LIN {X 0,Y 323.294,Z 676.092,A -85,B 0,C 180,E1 15567.964,E2 15567.964} C_VEL
LIN {X 0,Y 321.355,Z 689.746,A -85,B 0,C 180,E1 15566.345,E2 15566.345} C_VEL
LIN {X 0,Y 319.343,Z 702.477,A -85,B 0,C 180,E1 15564.432,E2 15564.432} C_VEL
LIN {X 0,Y 317.522,Z 713.237,A -85,B 0,C 180,E1 15562.402,E2 15562.402} C_VEL
LIN {X 0,Y 315.747,Z 723.463,A -85,B 0,C 180,E1 15559.972,E2 15559.972} C_VEL
LIN {X 0,Y 314.38,Z 731.614,A -85,B 0,C 180,E1 15557.512,E2 15557.512} C_VEL
LIN {X 0,Y 313.266,Z 738.806,A -85,B 0,C 180,E1 15554.64,E2 15554.64} C_VEL
LIN {X 0,Y 312.607,Z 743.939,A -85,B 0,C 180,E1 15551.797,E2 15551.797} C_VEL
LIN {X 0,Y 312.265,Z 747.451,A -85,B 0,C 180,E1 15548.715,E2 15548.715} C_VEL
LIN {X 0,Y 312.168,Z 749.028,A -85,B 0,C 180,E1 15545.799,E2 15545.799} C_VEL
LIN {X 0,Y 312.206,Z 748.828,A -85,B 0,C 180,E1 15542.747,E2 15542.747} C_VEL
LIN {X 0,Y 312.438,Z 746.912,A -85,B 0,C 180,E1 15539.776,E2 15539.776} C_VEL
LIN {X 0,Y 312.956,Z 743.159,A -85,B 0,C 180,E1 15536.833,E2 15536.833} C_VEL
LIN {X 0,Y 313.904,Z 737.534,A -85,B 0,C 180,E1 15533.898,E2 15533.898} C_VEL
LIN {X 0,Y 315.295,Z 730.063,A -85,B 0,C 180,E1 15531.108,E2 15531.108} C_VEL
LIN {X 0,Y 316.967,Z 721.566,A -85,B 0,C 180,E1 15528.658,E2 15528.658} C_VEL
LIN {X 0,Y 319.018,Z 711.003,A -85,B 0,C 180,E1 15526.287,E2 15526.287} C_VEL
LIN {X 0,Y 321.176,Z 699.388,A -85,B 0,C 180,E1 15524.215,E2 15524.215} C_VEL
LIN {X 0,Y 323.403,Z 686.141,A -85,B 0,C 180,E1 15522.365,E2 15522.365} C_VEL
LIN {X 0,Y 325.505,Z 671.84,A -85,B 0,C 180,E1 15520.801,E2 15520.801} C_VEL
LIN {X 0,Y 327.265,Z 657.03,A -85,B 0,C 180,E1 15519.581,E2 15519.581} C_VEL
LIN {X 0,Y 328.688,Z 641.061,A -85,B 0,C 180,E1 15518.618,E2 15518.618} C_VEL
LIN {X 0,Y 329.594,Z 624.254,A -85,B 0,C 180,E1 15517.968,E2 15517.968} C_VEL
LIN {X 0,Y 333.422,Z 501.812,A -85,B 0,C 180,E1 15515.207,E2 15515.207} C_VEL
LIN {X 0,Y 331.425,Z 482.705,A -85,B 0,C 180,E1 15514.449,E2 15514.449} C_VEL
LIN {X 0,Y 335.442,Z 437.528,A -85,B 0,C 180,E1 15509.848,E2 15509.848} C_VEL
LIN {X 0,Y 338.999,Z 399.053,A -85,B 0,C 180,E1 15505.967,E2 15505.967} C_VEL
LIN {X 0,Y 342.306,Z 362.127,A -85,B 0,C 180,E1 15502.249,E2 15502.249} C_VEL
LIN {X 0,Y 337.591,Z 346.974,A -85,B 0,C 180,E1 15499.734,E2 15499.734} C_VEL
LIN {X 0,Y 332.324,Z 333.278,A -85,B 0,C 180,E1 15497.149,E2 15497.149} C_VEL
LIN {X 0,Y 326.437,Z 320.297,A -85,B 0,C 180,E1 15494.366,E2 15494.366} C_VEL
LIN {X 0,Y 321.45,Z 310.966,A -85,B 0,C 180,E1 15492.029,E2 15492.029} C_VEL
LIN {X 0,Y 319.417,Z 307.063,A -85,B 0,C 180,E1 15491.009,E2 15491.009} C_VEL
LIN {X 0,Y 317.338,Z 303.417,A -85,B 0,C 180,E1 15489.98,E2 15489.98} C_VEL
LIN {X 0,Y 316.226,Z 301.786,A -85,B 0,C 180,E1 15489.464,E2 15489.464} C_VEL
LIN {X 0,Y 314.376,Z 298.507,A -85,B 0,C 180,E1 15488.478,E2 15488.478} C_VEL
LIN {X 0,Y 314.155,Z 297.393,A -85,B 0,C 180,E1 15487.959,E2 15487.959} C_VEL
LIN {X 0,Y 314.165,Z 297.347,A -85,B 0,C 180,E1 15483.467,E2 15483.467} C_VEL
LIN {X 0,Y 314.171,Z 297.344,A -85,B 0,C 180,E1 15479.089,E2 15479.089} C_VEL
LIN {X 0,Y 314.151,Z 297.354,A -85,B 0,C 180,E1 15474.522,E2 15474.522} C_VEL
LIN {X 0,Y 314.146,Z 297.345,A -85,B 0,C 180,E1 15470.104,E2 15470.104} C_VEL
LIN {X 0,Y 314.161,Z 297.354,A -85,B 0,C 180,E1 15465.627,E2 15465.627} C_VEL
LIN {X 0,Y 314.17,Z 297.343,A -85,B 0,C 180,E1 15461.251,E2 15461.251} C_VEL
LIN {X 0,Y 314.172,Z 297.351,A -85,B 0,C 180,E1 15456.758,E2 15456.758} C_VEL
LIN {X 0,Y 314.155,Z 297.349,A -85,B 0,C 180,E1 15452.22,E2 15452.22} C_VEL
LIN {X 0,Y 314.207,Z 297.632,A -85,B 0,C 180,E1 15448.543,E2 15448.543} C_VEL
LIN {X 0,Y 315.623,Z 301.081,A -85,B 0,C 180,E1 15447.631,E2 15447.631} C_VEL
LIN {X 0,Y 322.969,Z 317.218,A -85,B 0,C 180,E1 15443.751,E2 15443.751} C_VEL
LIN {X 0,Y 325.12,Z 321.958,A -85,B 0,C 180,E1 15442.766,E2 15442.766} C_VEL
LIN {X 0,Y 339.923,Z 346.539,A -85,B 0,C 180,E1 15439.593,E2 15439.593} C_VEL
LIN {X 0,Y 354.859,Z 373.04,A -85,B 0,C 180,E1 15436.679,E2 15436.679} C_VEL
LIN {X 0,Y 356.871,Z 377.15,A -85,B 0,C 180,E1 15436.291,E2 15436.291} C_VEL
LIN {X 0,Y 344.034,Z 576.734,A -85,B 0,C 180,E1 15431.093,E2 15431.093} C_VEL
LIN {X 0,Y 341.881,Z 598.232,A -85,B 0,C 180,E1 15430.243,E2 15430.243} C_VEL
LIN {X 0,Y 339.198,Z 619.151,A -85,B 0,C 180,E1 15429.107,E2 15429.107} C_VEL
LIN {X 0,Y 336.079,Z 639.65,A -85,B 0,C 180,E1 15427.655,E2 15427.655} C_VEL
LIN {X 0,Y 332.807,Z 658.657,A -85,B 0,C 180,E1 15425.966,E2 15425.966} C_VEL
LIN {X 0,Y 329.239,Z 677.46,A -85,B 0,C 180,E1 15423.908,E2 15423.908} C_VEL
LIN {X 0,Y 325.708,Z 695.046,A -85,B 0,C 180,E1 15421.558,E2 15421.558} C_VEL
LIN {X 0,Y 322.353,Z 711.252,A -85,B 0,C 180,E1 15418.936,E2 15418.936} C_VEL
LIN {X 0,Y 319.275,Z 726.233,A -85,B 0,C 180,E1 15416.001,E2 15416.001} C_VEL
LIN {X 0,Y 316.82,Z 738.788,A -85,B 0,C 180,E1 15413.035,E2 15413.035} C_VEL
LIN {X 0,Y 314.859,Z 749.859,A -85,B 0,C 180,E1 15409.861,E2 15409.861} C_VEL
LIN {X 0,Y 313.501,Z 758.929,A -85,B 0,C 180,E1 15406.679,E2 15406.679} C_VEL
LIN {X 0,Y 312.614,Z 766.626,A -85,B 0,C 180,E1 15403.312,E2 15403.312} C_VEL
LIN {X 0,Y 312.189,Z 772.809,A -85,B 0,C 180,E1 15399.771,E2 15399.771} C_VEL
LIN {X 0,Y 312.1,Z 776.968,A -85,B 0,C 180,E1 15396.436,E2 15396.436} C_VEL
LIN {X 0,Y 312.119,Z 779.473,A -85,B 0,C 180,E1 15393.12,E2 15393.12} C_VEL
LIN {X 0,Y 312.146,Z 780.41,A -85,B 0,C 180,E1 15389.814,E2 15389.814} C_VEL
LIN {X 0,Y 312.083,Z 779.858,A -85,B 0,C 180,E1 15386.508,E2 15386.508} C_VEL
LIN {X 0,Y 312.051,Z 777.77,A -85,B 0,C 180,E1 15383.189,E2 15383.189} C_VEL
LIN {X 0,Y 312.18,Z 774.12,A -85,B 0,C 180,E1 15379.852,E2 15379.852} C_VEL
LIN {X 0,Y 312.695,Z 768.613,A -85,B 0,C 180,E1 15376.311,E2 15376.311} C_VEL
LIN {X 0,Y 313.732,Z 761.756,A -85,B 0,C 180,E1 15372.948,E2 15372.948} C_VEL
LIN {X 0,Y 315.522,Z 752.593,A -85,B 0,C 180,E1 15369.404,E2 15369.404} C_VEL
LIN {X 0,Y 318.153,Z 741.278,A -85,B 0,C 180,E1 15365.884,E2 15365.884} C_VEL
LIN {X 0,Y 321.514,Z 728.328,A -85,B 0,C 180,E1 15362.595,E2 15362.595} C_VEL
LIN {X 0,Y 325.509,Z 713.816,A -85,B 0,C 180,E1 15359.546,E2 15359.546} C_VEL
LIN {X 0,Y 330.18,Z 697.464,A -85,B 0,C 180,E1 15356.697,E2 15356.697} C_VEL
LIN {X 0,Y 335.464,Z 679.029,A -85,B 0,C 180,E1 15354.042,E2 15354.042} C_VEL
LIN {X 0,Y 340.919,Z 659.877,A -85,B 0,C 180,E1 15351.768,E2 15351.768} C_VEL
LIN {X 0,Y 346.959,Z 638.42,A -85,B 0,C 180,E1 15349.686,E2 15349.686} C_VEL
LIN {X 0,Y 353.072,Z 616.191,A -85,B 0,C 180,E1 15347.951,E2 15347.951} C_VEL
LIN {X 0,Y 358.873,Z 594.337,A -85,B 0,C 180,E1 15346.623,E2 15346.623} C_VEL
LIN {X 0,Y 364.618,Z 570.64,A -85,B 0,C 180,E1 15345.534,E2 15345.534} C_VEL
LIN {X 0,Y 377.031,Z 516.92,A -85,B 0,C 180,E1 15343.532,E2 15343.532} C_VEL
LIN {X 0,Y 381.467,Z 500.047,A -85,B 0,C 180,E1 15342.895,E2 15342.895} C_VEL
LIN {X 0,Y 366.445,Z 559.755,A -85,B 0,C 180,E1 15340.585,E2 15340.585} C_VEL
LIN {X 0,Y 360.935,Z 581.963,A -85,B 0,C 180,E1 15339.579,E2 15339.579} C_VEL
LIN {X 0,Y 355.075,Z 603.113,A -85,B 0,C 180,E1 15338.279,E2 15338.279} C_VEL
LIN {X 0,Y 348.859,Z 624.354,A -85,B 0,C 180,E1 15336.594,E2 15336.594} C_VEL
LIN {X 0,Y 342.955,Z 643.935,A -85,B 0,C 180,E1 15334.646,E2 15334.646} C_VEL
LIN {X 0,Y 337.175,Z 662.515,A -85,B 0,C 180,E1 15332.361,E2 15332.361} C_VEL
LIN {X 0,Y 331.809,Z 679.598,A -85,B 0,C 180,E1 15329.788,E2 15329.788} C_VEL
LIN {X 0,Y 327.161,Z 694.304,A -85,B 0,C 180,E1 15327.088,E2 15327.088} C_VEL
LIN {X 0,Y 323.006,Z 707.545,A -85,B 0,C 180,E1 15324.117,E2 15324.117} C_VEL
LIN {X 0,Y 319.633,Z 718.492,A -85,B 0,C 180,E1 15321.083,E2 15321.083} C_VEL
LIN {X 0,Y 316.864,Z 727.897,A -85,B 0,C 180,E1 15317.823,E2 15317.823} C_VEL
LIN {X 0,Y 314.86,Z 735.32,A -85,B 0,C 180,E1 15314.528,E2 15314.528} C_VEL
LIN {X 0,Y 313.523,Z 740.919,A -85,B 0,C 180,E1 15311.217,E2 15311.217} C_VEL
LIN {X 0,Y 312.721,Z 744.807,A -85,B 0,C 180,E1 15307.902,E2 15307.902} C_VEL
LIN {X 0,Y 312.307,Z 747.109,A -85,B 0,C 180,E1 15304.406,E2 15304.406} C_VEL
LIN {X 0,Y 312.167,Z 747.631,A -85,B 0,C 180,E1 15301.101,E2 15301.101} C_VEL
LIN {X 0,Y 312.123,Z 746.506,A -85,B 0,C 180,E1 15297.796,E2 15297.796} C_VEL
LIN {X 0,Y 312.205,Z 743.731,A -85,B 0,C 180,E1 15294.486,E2 15294.486} C_VEL
LIN {X 0,Y 312.502,Z 739.236,A -85,B 0,C 180,E1 15291.165,E2 15291.165} C_VEL
LIN {X 0,Y 313.109,Z 733.292,A -85,B 0,C 180,E1 15288.02,E2 15288.02} C_VEL
LIN {X 0,Y 314.157,Z 725.57,A -85,B 0,C 180,E1 15284.871,E2 15284.871} C_VEL
LIN {X 0,Y 315.737,Z 715.857,A -85,B 0,C 180,E1 15281.728,E2 15281.728} C_VEL
LIN {X 0,Y 317.776,Z 704.613,A -85,B 0,C 180,E1 15278.786,E2 15278.786} C_VEL
LIN {X 0,Y 320.217,Z 691.886,A -85,B 0,C 180,E1 15276.051,E2 15276.051} C_VEL
LIN {X 0,Y 322.985,Z 677.669,A -85,B 0,C 180,E1 15273.526,E2 15273.526} C_VEL
LIN {X 0,Y 325.992,Z 661.889,A -85,B 0,C 180,E1 15271.213,E2 15271.213} C_VEL
LIN {X 0,Y 329.153,Z 644.286,A -85,B 0,C 180,E1 15269.111,E2 15269.111} C_VEL
LIN {X 0,Y 332.082,Z 626.513,A -85,B 0,C 180,E1 15267.387,E2 15267.387} C_VEL
LIN {X 0,Y 334.806,Z 607.979,A -85,B 0,C 180,E1 15265.947,E2 15265.947} C_VEL
LIN {X 0,Y 337.196,Z 588.684,A -85,B 0,C 180,E1 15264.778,E2 15264.778} C_VEL
LIN {X 0,Y 339.329,Z 567.504,A -85,B 0,C 180,E1 15263.841,E2 15263.841} C_VEL
LIN {X 0,Y 341.441,Z 536.028,A -85,B 0,C 180,E1 15262.91,E2 15262.91} C_VEL
LIN {X 0,Y 351.309,Z 385.374,A -85,B 0,C 180,E1 15258.813,E2 15258.813} C_VEL
LIN {X 0,Y 349.678,Z 373.169,A -85,B 0,C 180,E1 15258.18,E2 15258.18} C_VEL
LIN {X 0,Y 335.154,Z 345.914,A -85,B 0,C 180,E1 15255.269,E2 15255.269} C_VEL
LIN {X 0,Y 330.764,Z 337.858,A -85,B 0,C 180,E1 15254.291,E2 15254.291} C_VEL
LIN {X 0,Y 323.739,Z 320.175,A -85,B 0,C 180,E1 15250.436,E2 15250.436} C_VEL
LIN {X 0,Y 317.35,Z 304.98,A -85,B 0,C 180,E1 15246.773,E2 15246.773} C_VEL
LIN {X 0,Y 314.204,Z 297.608,A -85,B 0,C 180,E1 15244.813,E2 15244.813} C_VEL
LIN {X 0,Y 314.174,Z 297.326,A -85,B 0,C 180,E1 15240.401,E2 15240.401} C_VEL
LIN {X 0,Y 314.192,Z 297.569,A -85,B 0,C 180,E1 15238.826,E2 15238.826} C_VEL
LIN {X 0,Y 315.268,Z 300.467,A -85,B 0,C 180,E1 15238.154,E2 15238.154} C_VEL
LIN {X 0,Y 316.442,Z 302.54,A -85,B 0,C 180,E1 15237.678,E2 15237.678} C_VEL
LIN {X 0,Y 323.43,Z 317.197,A -85,B 0,C 180,E1 15234.647,E2 15234.647} C_VEL
LIN {X 0,Y 330.61,Z 334.343,A -85,B 0,C 180,E1 15231.467,E2 15231.467} C_VEL
LIN {X 0,Y 336.995,Z 352.041,A -85,B 0,C 180,E1 15228.512,E2 15228.512} C_VEL
LIN {X 0,Y 339.833,Z 361.857,A -85,B 0,C 180,E1 15227.014,E2 15227.014} C_VEL
LIN {X 0,Y 336.205,Z 402.075,A -85,B 0,C 180,E1 15222.89,E2 15222.89} C_VEL
LIN {X 0,Y 332.629,Z 441.744,A -85,B 0,C 180,E1 15218.82,E2 15218.82} C_VEL
LIN {X 0,Y 329.266,Z 482.332,A -85,B 0,C 180,E1 15214.683,E2 15214.683} C_VEL
LIN {X 0,Y 331.319,Z 504.222,A -85,B 0,C 180,E1 15213.952,E2 15213.952} C_VEL
LIN {X 0,Y 327.654,Z 626.241,A -85,B 0,C 180,E1 15211.226,E2 15211.226} C_VEL
LIN {X 0,Y 327.484,Z 629.952,A -85,B 0,C 180,E1 15211.095,E2 15211.095} C_VEL
LIN {X 0,Y 325.817,Z 638.541,A -85,B 0,C 180,E1 15210.832,E2 15210.832} C_VEL
LIN {X 0,Y 319.849,Z 653.981,A -85,B 0,C 180,E1 15210.329,E2 15210.329} C_VEL
LIN {X 0,Y 317.824,Z 661.131,A -85,B 0,C 180,E1 15209.901,E2 15209.901} C_VEL
LIN {X 0,Y 317.518,Z 663.107,A -85,B 0,C 180,E1 15209.745,E2 15209.745} C_VEL
LIN {X 0,Y 315.7,Z 677.597,A -85,B 0,C 180,E1 15208.369,E2 15208.369} C_VEL
LIN {X 0,Y 313.688,Z 691.008,A -85,B 0,C 180,E1 15206.713,E2 15206.713} C_VEL
LIN {X 0,Y 311.602,Z 703.615,A -85,B 0,C 180,E1 15204.751,E2 15204.751} C_VEL
LIN {X 0,Y 309.591,Z 714.862,A -85,B 0,C 180,E1 15202.527,E2 15202.527} C_VEL
LIN {X 0,Y 307.812,Z 724.685,A -85,B 0,C 180,E1 15200.089,E2 15200.089} C_VEL
LIN {X 0,Y 306.314,Z 733.152,A -85,B 0,C 180,E1 15197.37,E2 15197.37} C_VEL
LIN {X 0,Y 305.271,Z 739.69,A -85,B 0,C 180,E1 15194.618,E2 15194.618} C_VEL
LIN {X 0,Y 304.625,Z 744.461,A -85,B 0,C 180,E1 15191.834,E2 15191.834} C_VEL
LIN {X 0,Y 304.281,Z 747.806,A -85,B 0,C 180,E1 15188.813,E2 15188.813} C_VEL
LIN {X 0,Y 304.177,Z 749.381,A -85,B 0,C 180,E1 15185.948,E2 15185.948} C_VEL
LIN {X 0,Y 304.209,Z 749.326,A -85,B 0,C 180,E1 15182.964,E2 15182.964} C_VEL
LIN {X 0,Y 304.444,Z 747.509,A -85,B 0,C 180,E1 15179.838,E2 15179.838} C_VEL
LIN {X 0,Y 304.981,Z 743.907,A -85,B 0,C 180,E1 15176.807,E2 15176.807} C_VEL
LIN {X 0,Y 305.985,Z 738.311,A -85,B 0,C 180,E1 15173.743,E2 15173.743} C_VEL
LIN {X 0,Y 307.351,Z 731.431,A -85,B 0,C 180,E1 15171.034,E2 15171.034} C_VEL
LIN {X 0,Y 309.223,Z 722.437,A -85,B 0,C 180,E1 15168.326,E2 15168.326} C_VEL
LIN {X 0,Y 311.258,Z 712.593,A -85,B 0,C 180,E1 15166.019,E2 15166.019} C_VEL
LIN {X 0,Y 313.635,Z 700.469,A -85,B 0,C 180,E1 15163.773,E2 15163.773} C_VEL
LIN {X 0,Y 315.884,Z 687.906,A -85,B 0,C 180,E1 15161.944,E2 15161.944} C_VEL
LIN {X 0,Y 318.138,Z 673.471,A -85,B 0,C 180,E1 15160.298,E2 15160.298} C_VEL
LIN {X 0,Y 320.016,Z 658.803,A -85,B 0,C 180,E1 15159.031,E2 15159.031} C_VEL
LIN {X 0,Y 321.584,Z 642.411,A -85,B 0,C 180,E1 15157.998,E2 15157.998} C_VEL
LIN {X 0,Y 322.547,Z 626.195,A -85,B 0,C 180,E1 15157.332,E2 15157.332} C_VEL
LIN {X 0,Y 326.646,Z 502.725,A -85,B 0,C 180,E1 15154.479,E2 15154.479} C_VEL
LIN {X 0,Y 324.633,Z 483.021,A -85,B 0,C 180,E1 15153.67,E2 15153.67} C_VEL
LIN {X 0,Y 328.77,Z 438.859,A -85,B 0,C 180,E1 15149.118,E2 15149.118} C_VEL
LIN {X 0,Y 332.769,Z 398.4,A -85,B 0,C 180,E1 15144.971,E2 15144.971} C_VEL
LIN {X 0,Y 335.797,Z 365.098,A -85,B 0,C 180,E1 15141.576,E2 15141.576} C_VEL
LIN {X 0,Y 331.194,Z 350.272,A -85,B 0,C 180,E1 15139.03,E2 15139.03} C_VEL
LIN {X 0,Y 326.01,Z 336.794,A -85,B 0,C 180,E1 15136.39,E2 15136.39} C_VEL
LIN {X 0,Y 320.64,Z 324.896,A -85,B 0,C 180,E1 15133.71,E2 15133.71} C_VEL
LIN {X 0,Y 316.472,Z 316.888,A -85,B 0,C 180,E1 15131.661,E2 15131.661} C_VEL
LIN {X 0,Y 314.082,Z 312.525,A -85,B 0,C 180,E1 15130.455,E2 15130.455} C_VEL
LIN {X 0,Y 311.75,Z 308.29,A -85,B 0,C 180,E1 15129.229,E2 15129.229} C_VEL
LIN {X 0,Y 309.749,Z 304.971,A -85,B 0,C 180,E1 15128.166,E2 15128.166} C_VEL
LIN {X 0,Y 308.797,Z 303.284,A -85,B 0,C 180,E1 15127.629,E2 15127.629} C_VEL
LIN {X 0,Y 306.75,Z 300.399,A -85,B 0,C 180,E1 15126.551,E2 15126.551} C_VEL
LIN {X 0,Y 306.26,Z 298.675,A -85,B 0,C 180,E1 15125.997,E2 15125.997} C_VEL
LIN {X 0,Y 306.207,Z 298.337,A -85,B 0,C 180,E1 15124.12,E2 15124.12} C_VEL
LIN {X 0,Y 306.224,Z 298.337,A -85,B 0,C 180,E1 15119.627,E2 15119.627} C_VEL
LIN {X 0,Y 306.231,Z 298.337,A -85,B 0,C 180,E1 15115.131,E2 15115.131} C_VEL
LIN {X 0,Y 306.222,Z 298.333,A -85,B 0,C 180,E1 15110.794,E2 15110.794} C_VEL
LIN {X 0,Y 306.208,Z 298.34,A -85,B 0,C 180,E1 15106.211,E2 15106.211} C_VEL
LIN {X 0,Y 306.215,Z 298.335,A -85,B 0,C 180,E1 15101.733,E2 15101.733} C_VEL
LIN {X 0,Y 306.244,Z 298.334,A -85,B 0,C 180,E1 15097.138,E2 15097.138} C_VEL
LIN {X 0,Y 306.226,Z 298.335,A -85,B 0,C 180,E1 15092.589,E2 15092.589} C_VEL
LIN {X 0,Y 306.246,Z 298.564,A -85,B 0,C 180,E1 15089.96,E2 15089.96} C_VEL
LIN {X 0,Y 307.852,Z 302.276,A -85,B 0,C 180,E1 15088.909,E2 15088.909} C_VEL
LIN {X 0,Y 315.057,Z 318.13,A -85,B 0,C 180,E1 15084.942,E2 15084.942} C_VEL
LIN {X 0,Y 316.939,Z 322.177,A -85,B 0,C 180,E1 15084.072,E2 15084.072} C_VEL
LIN {X 0,Y 332.048,Z 347.169,A -85,B 0,C 180,E1 15080.693,E2 15080.693} C_VEL
LIN {X 0,Y 347.478,Z 374.403,A -85,B 0,C 180,E1 15077.564,E2 15077.564} C_VEL
LIN {X 0,Y 350.314,Z 380.038,A -85,B 0,C 180,E1 15077.007,E2 15077.007} C_VEL
LIN {X 0,Y 337.058,Z 576.643,A -85,B 0,C 180,E1 15071.753,E2 15071.753} C_VEL
LIN {X 0,Y 334.887,Z 597.608,A -85,B 0,C 180,E1 15070.911,E2 15070.911} C_VEL
LIN {X 0,Y 332.084,Z 618.839,A -85,B 0,C 180,E1 15069.738,E2 15069.738} C_VEL
LIN {X 0,Y 328.838,Z 639.488,A -85,B 0,C 180,E1 15068.247,E2 15068.247} C_VEL
LIN {X 0,Y 325.379,Z 658.903,A -85,B 0,C 180,E1 15066.482,E2 15066.482} C_VEL
LIN {X 0,Y 321.792,Z 677.22,A -85,B 0,C 180,E1 15064.434,E2 15064.434} C_VEL
LIN {X 0,Y 318.199,Z 694.568,A -85,B 0,C 180,E1 15062.073,E2 15062.073} C_VEL
LIN {X 0,Y 314.704,Z 710.893,A -85,B 0,C 180,E1 15059.38,E2 15059.38} C_VEL
LIN {X 0,Y 311.588,Z 725.552,A -85,B 0,C 180,E1 15056.456,E2 15056.456} C_VEL
LIN {X 0,Y 308.91,Z 738.785,A -85,B 0,C 180,E1 15053.256,E2 15053.256} C_VEL
LIN {X 0,Y 306.797,Z 750.422,A -85,B 0,C 180,E1 15049.81,E2 15049.81} C_VEL
LIN {X 0,Y 305.379,Z 759.821,A -85,B 0,C 180,E1 15046.352,E2 15046.352} C_VEL
LIN {X 0,Y 304.527,Z 767.412,A -85,B 0,C 180,E1 15042.803,E2 15042.803} C_VEL
LIN {X 0,Y 304.178,Z 772.851,A -85,B 0,C 180,E1 15039.458,E2 15039.458} C_VEL
LIN {X 0,Y 304.115,Z 776.821,A -85,B 0,C 180,E1 15036.037,E2 15036.037} C_VEL
LIN {X 0,Y 304.142,Z 779.211,A -85,B 0,C 180,E1 15032.636,E2 15032.636} C_VEL
LIN {X 0,Y 304.153,Z 779.937,A -85,B 0,C 180,E1 15029.433,E2 15029.433} C_VEL
LIN {X 0,Y 304.087,Z 779.271,A -85,B 0,C 180,E1 15026.039,E2 15026.039} C_VEL
LIN {X 0,Y 304.051,Z 777.109,A -85,B 0,C 180,E1 15022.63,E2 15022.63} C_VEL
LIN {X 0,Y 304.261,Z 773.101,A -85,B 0,C 180,E1 15019.01,E2 15019.01} C_VEL
LIN {X 0,Y 304.947,Z 767.241,A -85,B 0,C 180,E1 15015.293,E2 15015.293} C_VEL
LIN {X 0,Y 306.34,Z 759.409,A -85,B 0,C 180,E1 15011.541,E2 15011.541} C_VEL
LIN {X 0,Y 308.517,Z 749.839,A -85,B 0,C 180,E1 15007.916,E2 15007.916} C_VEL
LIN {X 0,Y 311.541,Z 738.368,A -85,B 0,C 180,E1 15004.4,E2 15004.4} C_VEL
LIN {X 0,Y 315.243,Z 725.575,A -85,B 0,C 180,E1 15001.176,E2 15001.176} C_VEL
LIN {X 0,Y 319.739,Z 710.854,A -85,B 0,C 180,E1 14998.095,E2 14998.095} C_VEL
LIN {X 0,Y 324.84,Z 694.576,A -85,B 0,C 180,E1 14995.267,E2 14995.267} C_VEL
LIN {X 0,Y 330.567,Z 676.536,A -85,B 0,C 180,E1 14992.665,E2 14992.665} C_VEL
LIN {X 0,Y 337.026,Z 656.216,A -85,B 0,C 180,E1 14990.257,E2 14990.257} C_VEL
LIN {X 0,Y 343.944,Z 634.344,A -85,B 0,C 180,E1 14988.15,E2 14988.15} C_VEL
LIN {X 0,Y 350.733,Z 612.655,A -85,B 0,C 180,E1 14986.49,E2 14986.49} C_VEL
LIN {X 0,Y 357.072,Z 591.467,A -85,B 0,C 180,E1 14985.23,E2 14985.23} C_VEL
LIN {X 0,Y 363.788,Z 566.83,A -85,B 0,C 180,E1 14984.134,E2 14984.134} C_VEL
LIN {X 0,Y 372.301,Z 533.607,A -85,B 0,C 180,E1 14982.874,E2 14982.874} C_VEL
LIN {X 0,Y 360.852,Z 576.04,A -85,B 0,C 180,E1 14981.152,E2 14981.152} C_VEL
LIN {X 0,Y 354.598,Z 596.497,A -85,B 0,C 180,E1 14980.007,E2 14980.007} C_VEL
LIN {X 0,Y 347.835,Z 617.125,A -85,B 0,C 180,E1 14978.486,E2 14978.486} C_VEL
LIN {X 0,Y 341.059,Z 637.015,A -85,B 0,C 180,E1 14976.625,E2 14976.625} C_VEL
LIN {X 0,Y 334.362,Z 656.332,A -85,B 0,C 180,E1 14974.375,E2 14974.375} C_VEL
LIN {X 0,Y 328.316,Z 673.71,A -85,B 0,C 180,E1 14971.895,E2 14971.895} C_VEL
LIN {X 0,Y 322.738,Z 689.716,A -85,B 0,C 180,E1 14969.103,E2 14969.103} C_VEL
LIN {X 0,Y 317.877,Z 703.571,A -85,B 0,C 180,E1 14966.126,E2 14966.126} C_VEL
LIN {X 0,Y 313.881,Z 715.175,A -85,B 0,C 180,E1 14963.067,E2 14963.067} C_VEL
LIN {X 0,Y 310.524,Z 725.268,A -85,B 0,C 180,E1 14959.76,E2 14959.76} C_VEL
LIN {X 0,Y 308.003,Z 733.339,A -85,B 0,C 180,E1 14956.404,E2 14956.404} C_VEL
LIN {X 0,Y 306.161,Z 739.845,A -85,B 0,C 180,E1 14952.83,E2 14952.83} C_VEL
LIN {X 0,Y 305.03,Z 744.424,A -85,B 0,C 180,E1 14949.242,E2 14949.242} C_VEL
LIN {X 0,Y 304.445,Z 747.163,A -85,B 0,C 180,E1 14945.654,E2 14945.654} C_VEL
LIN {X 0,Y 304.206,Z 748.1,A -85,B 0,C 180,E1 14942.26,E2 14942.26} C_VEL
LIN {X 0,Y 304.14,Z 747.413,A -85,B 0,C 180,E1 14938.869,E2 14938.869} C_VEL
LIN {X 0,Y 304.167,Z 745.086,A -85,B 0,C 180,E1 14935.474,E2 14935.474} C_VEL
LIN {X 0,Y 304.381,Z 741.334,A -85,B 0,C 180,E1 14932.259,E2 14932.259} C_VEL
LIN {X 0,Y 304.928,Z 735.584,A -85,B 0,C 180,E1 14928.844,E2 14928.844} C_VEL
LIN {X 0,Y 305.866,Z 728.363,A -85,B 0,C 180,E1 14925.614,E2 14925.614} C_VEL
LIN {X 0,Y 307.335,Z 719.193,A -85,B 0,C 180,E1 14922.388,E2 14922.388} C_VEL
LIN {X 0,Y 309.278,Z 708.546,A -85,B 0,C 180,E1 14919.366,E2 14919.366} C_VEL
LIN {X 0,Y 311.636,Z 696.489,A -85,B 0,C 180,E1 14916.556,E2 14916.556} C_VEL
LIN {X 0,Y 314.332,Z 683.05,A -85,B 0,C 180,E1 14913.961,E2 14913.961} C_VEL
LIN {X 0,Y 317.368,Z 667.769,A -85,B 0,C 180,E1 14911.523,E2 14911.523} C_VEL
LIN {X 0,Y 320.536,Z 651.099,A -85,B 0,C 180,E1 14909.335,E2 14909.335} C_VEL
LIN {X 0,Y 323.76,Z 632.878,A -85,B 0,C 180,E1 14907.39,E2 14907.39} C_VEL
LIN {X 0,Y 326.7,Z 614.266,A -85,B 0,C 180,E1 14905.795,E2 14905.795} C_VEL
LIN {X 0,Y 329.424,Z 594.374,A -85,B 0,C 180,E1 14904.462,E2 14904.462} C_VEL
LIN {X 0,Y 331.752,Z 573.477,A -85,B 0,C 180,E1 14903.416,E2 14903.416} C_VEL
LIN {X 0,Y 333.538,Z 551.332,A -85,B 0,C 180,E1 14902.664,E2 14902.664} C_VEL
LIN {X 0,Y 344.781,Z 386.537,A -85,B 0,C 180,E1 14898.062,E2 14898.062} C_VEL
LIN {X 0,Y 343.509,Z 376.898,A -85,B 0,C 180,E1 14897.552,E2 14897.552} C_VEL
LIN {X 0,Y 329.817,Z 350.976,A -85,B 0,C 180,E1 14894.726,E2 14894.726} C_VEL
LIN {X 0,Y 322.394,Z 337.465,A -85,B 0,C 180,E1 14893.025,E2 14893.025} C_VEL
LIN {X 0,Y 315.826,Z 320.992,A -85,B 0,C 180,E1 14889.286,E2 14889.286} C_VEL
LIN {X 0,Y 309.267,Z 305.717,A -85,B 0,C 180,E1 14885.439,E2 14885.439} C_VEL
LIN {X 0,Y 306.256,Z 298.499,A -85,B 0,C 180,E1 14883.427,E2 14883.427} C_VEL
LIN {X 0,Y 306.266,Z 298.491,A -85,B 0,C 180,E1 14880.239,E2 14880.239} C_VEL
LIN {X 0,Y 306.625,Z 299.95,A -85,B 0,C 180,E1 14879.842,E2 14879.842} C_VEL
LIN {X 0,Y 308.818,Z 304.202,A -85,B 0,C 180,E1 14878.845,E2 14878.845} C_VEL
LIN {X 0,Y 315.036,Z 316.957,A -85,B 0,C 180,E1 14876.078,E2 14876.078} C_VEL
LIN {X 0,Y 321.803,Z 332.294,A -85,B 0,C 180,E1 14873.049,E2 14873.049} C_VEL
LIN {X 0,Y 328.534,Z 350.253,A -85,B 0,C 180,E1 14869.877,E2 14869.877} C_VEL
LIN {X 0,Y 332.994,Z 364.788,A -85,B 0,C 180,E1 14867.565,E2 14867.565} C_VEL
LIN {X 0,Y 328.99,Z 407.138,A -85,B 0,C 180,E1 14863.177,E2 14863.177} C_VEL
LIN {X 0,Y 324.968,Z 450.502,A -85,B 0,C 180,E1 14858.673,E2 14858.673} C_VEL
LIN {X 0,Y 322.15,Z 482.695,A -85,B 0,C 180,E1 14855.35,E2 14855.35} C_VEL
LIN {X 0,Y 324.203,Z 504.951,A -85,B 0,C 180,E1 14854.584,E2 14854.584} C_VEL
LIN {X 0,Y 320.395,Z 626.529,A -85,B 0,C 180,E1 14851.818,E2 14851.818} C_VEL
LIN {X 0,Y 319.442,Z 642.663,A -85,B 0,C 180,E1 14851.126,E2 14851.126} C_VEL
LIN {X 0,Y 318.04,Z 658.371,A -85,B 0,C 180,E1 14850.122,E2 14850.122} C_VEL
LIN {X 0,Y 317.518,Z 663.107,A -85,B 0,C 180,E1 14849.745,E2 14849.745} C_VEL
LIN {X 0,Y 315.774,Z 670.088,A -85,B 0,C 180,E1 14849.203,E2 14849.203} C_VEL
LIN {X 0,Y 309.07,Z 684.144,A -85,B 0,C 180,E1 14848.045,E2 14848.045} C_VEL
LIN {X 0,Y 306.269,Z 691.31,A -85,B 0,C 180,E1 14847.222,E2 14847.222} C_VEL
LIN {X 0,Y 305.895,Z 693.038,A -85,B 0,C 180,E1 14846.982,E2 14846.982} C_VEL
LIN {X 0,Y 303.776,Z 705.14,A -85,B 0,C 180,E1 14844.998,E2 14844.998} C_VEL
LIN {X 0,Y 301.589,Z 716.836,A -85,B 0,C 180,E1 14842.573,E2 14842.573} C_VEL
LIN {X 0,Y 299.746,Z 726.488,A -85,B 0,C 180,E1 14840.013,E2 14840.013} C_VEL
LIN {X 0,Y 298.247,Z 734.68,A -85,B 0,C 180,E1 14837.219,E2 14837.219} C_VEL
LIN {X 0,Y 297.213,Z 740.914,A -85,B 0,C 180,E1 14834.39,E2 14834.39} C_VEL
LIN {X 0,Y 296.555,Z 745.698,A -85,B 0,C 180,E1 14831.321,E2 14831.321} C_VEL
LIN {X 0,Y 296.269,Z 748.563,A -85,B 0,C 180,E1 14828.419,E2 14828.419} C_VEL
LIN {X 0,Y 296.18,Z 749.881,A -85,B 0,C 180,E1 14825.247,E2 14825.247} C_VEL
LIN {X 0,Y 296.259,Z 749.494,A -85,B 0,C 180,E1 14822.16,E2 14822.16} C_VEL
LIN {X 0,Y 296.546,Z 747.466,A -85,B 0,C 180,E1 14819.173,E2 14819.173} C_VEL
LIN {X 0,Y 297.199,Z 743.571,A -85,B 0,C 180,E1 14816.053,E2 14816.053} C_VEL
LIN {X 0,Y 298.269,Z 738.131,A -85,B 0,C 180,E1 14813.13,E2 14813.13} C_VEL
LIN {X 0,Y 299.875,Z 730.609,A -85,B 0,C 180,E1 14810.198,E2 14810.198} C_VEL
LIN {X 0,Y 301.777,Z 722.054,A -85,B 0,C 180,E1 14807.635,E2 14807.635} C_VEL
LIN {X 0,Y 304.089,Z 711.402,A -85,B 0,C 180,E1 14805.151,E2 14805.151} C_VEL
LIN {X 0,Y 306.506,Z 699.659,A -85,B 0,C 180,E1 14802.984,E2 14802.984} C_VEL
LIN {X 0,Y 308.971,Z 686.351,A -85,B 0,C 180,E1 14801.065,E2 14801.065} C_VEL
LIN {X 0,Y 311.195,Z 672.566,A -85,B 0,C 180,E1 14799.508,E2 14799.508} C_VEL
LIN {X 0,Y 313.132,Z 657.699,A -85,B 0,C 180,E1 14798.237,E2 14798.237} C_VEL
LIN {X 0,Y 314.68,Z 641.854,A -85,B 0,C 180,E1 14797.247,E2 14797.247} C_VEL
LIN {X 0,Y 315.684,Z 624.99,A -85,B 0,C 180,E1 14796.57,E2 14796.57} C_VEL
LIN {X 0,Y 319.916,Z 503.512,A -85,B 0,C 180,E1 14793.715,E2 14793.715} C_VEL
LIN {X 0,Y 317.902,Z 483.756,A -85,B 0,C 180,E1 14792.89,E2 14792.89} C_VEL
LIN {X 0,Y 322.289,Z 439.065,A -85,B 0,C 180,E1 14788.234,E2 14788.234} C_VEL
LIN {X 0,Y 326.267,Z 400.494,A -85,B 0,C 180,E1 14784.246,E2 14784.246} C_VEL
LIN {X 0,Y 329.455,Z 368.511,A -85,B 0,C 180,E1 14780.939,E2 14780.939} C_VEL
LIN {X 0,Y 324.873,Z 353.638,A -85,B 0,C 180,E1 14778.297,E2 14778.297} C_VEL
LIN {X 0,Y 319.801,Z 340.408,A -85,B 0,C 180,E1 14775.598,E2 14775.598} C_VEL
LIN {X 0,Y 314.261,Z 327.976,A -85,B 0,C 180,E1 14772.682,E2 14772.682} C_VEL
LIN {X 0,Y 309.222,Z 318.517,A -85,B 0,C 180,E1 14770.056,E2 14770.056} C_VEL
LIN {X 0,Y 306.971,Z 314.379,A -85,B 0,C 180,E1 14768.807,E2 14768.807} C_VEL
LIN {X 0,Y 304.436,Z 309.854,A -85,B 0,C 180,E1 14767.36,E2 14767.36} C_VEL
LIN {X 0,Y 302.17,Z 306.458,A -85,B 0,C 180,E1 14766.079,E2 14766.079} C_VEL
LIN {X 0,Y 301.328,Z 304.672,A -85,B 0,C 180,E1 14765.496,E2 14765.496} C_VEL
LIN {X 0,Y 299.045,Z 301.904,A -85,B 0,C 180,E1 14764.219,E2 14764.219} C_VEL
LIN {X 0,Y 298.345,Z 299.72,A -85,B 0,C 180,E1 14763.459,E2 14763.459} C_VEL
LIN {X 0,Y 298.266,Z 299.329,A -85,B 0,C 180,E1 14762.306,E2 14762.306} C_VEL
LIN {X 0,Y 298.272,Z 299.329,A -85,B 0,C 180,E1 14757.887,E2 14757.887} C_VEL
LIN {X 0,Y 298.3,Z 299.319,A -85,B 0,C 180,E1 14753.263,E2 14753.263} C_VEL
LIN {X 0,Y 298.284,Z 299.331,A -85,B 0,C 180,E1 14748.79,E2 14748.79} C_VEL
LIN {X 0,Y 298.27,Z 299.322,A -85,B 0,C 180,E1 14744.16,E2 14744.16} C_VEL
LIN {X 0,Y 298.281,Z 299.332,A -85,B 0,C 180,E1 14739.598,E2 14739.598} C_VEL
LIN {X 0,Y 298.292,Z 299.323,A -85,B 0,C 180,E1 14735.23,E2 14735.23} C_VEL
LIN {X 0,Y 298.325,Z 299.565,A -85,B 0,C 180,E1 14731.41,E2 14731.41} C_VEL
LIN {X 0,Y 301.597,Z 307.018,A -85,B 0,C 180,E1 14729.301,E2 14729.301} C_VEL
LIN {X 0,Y 307.776,Z 320.683,A -85,B 0,C 180,E1 14725.805,E2 14725.805} C_VEL
LIN {X 0,Y 309.708,Z 324.106,A -85,B 0,C 180,E1 14725.179,E2 14725.179} C_VEL
LIN {X 0,Y 322.915,Z 345.738,A -85,B 0,C 180,E1 14722.104,E2 14722.104} C_VEL
LIN {X 0,Y 337.2,Z 370.561,A -85,B 0,C 180,E1 14719.058,E2 14719.058} C_VEL
LIN {X 0,Y 343.751,Z 382.926,A -85,B 0,C 180,E1 14717.735,E2 14717.735} C_VEL
LIN {X 0,Y 330.104,Z 576.48,A -85,B 0,C 180,E1 14712.434,E2 14712.434} C_VEL
LIN {X 0,Y 327.862,Z 597.383,A -85,B 0,C 180,E1 14711.576,E2 14711.576} C_VEL
LIN {X 0,Y 324.939,Z 618.799,A -85,B 0,C 180,E1 14710.367,E2 14710.367} C_VEL
LIN {X 0,Y 321.68,Z 638.915,A -85,B 0,C 180,E1 14708.89,E2 14708.89} C_VEL
LIN {X 0,Y 318.143,Z 658.191,A -85,B 0,C 180,E1 14707.112,E2 14707.112} C_VEL
LIN {X 0,Y 314.434,Z 676.579,A -85,B 0,C 180,E1 14705.024,E2 14705.024} C_VEL
LIN {X 0,Y 310.714,Z 693.994,A -85,B 0,C 180,E1 14702.613,E2 14702.613} C_VEL
LIN {X 0,Y 307.104,Z 710.311,A -85,B 0,C 180,E1 14699.874,E2 14699.874} C_VEL
LIN {X 0,Y 303.92,Z 724.797,A -85,B 0,C 180,E1 14696.932,E2 14696.932} C_VEL
LIN {X 0,Y 301.149,Z 738,A -85,B 0,C 180,E1 14693.684,E2 14693.684} C_VEL
LIN {X 0,Y 299.039,Z 749.118,A -85,B 0,C 180,E1 14690.346,E2 14690.346} C_VEL
LIN {X 0,Y 297.581,Z 758.21,A -85,B 0,C 180,E1 14686.994,E2 14686.994} C_VEL
LIN {X 0,Y 296.642,Z 765.905,A -85,B 0,C 180,E1 14683.446,E2 14683.446} C_VEL
LIN {X 0,Y 296.206,Z 772.062,A -85,B 0,C 180,E1 14679.714,E2 14679.714} C_VEL
LIN {X 0,Y 296.13,Z 776.162,A -85,B 0,C 180,E1 14676.2,E2 14676.2} C_VEL
LIN {X 0,Y 296.158,Z 778.504,A -85,B 0,C 180,E1 14672.901,E2 14672.901} C_VEL
LIN {X 0,Y 296.169,Z 779.439,A -85,B 0,C 180,E1 14669.418,E2 14669.418} C_VEL
LIN {X 0,Y 296.093,Z 778.868,A -85,B 0,C 180,E1 14665.931,E2 14665.931} C_VEL
LIN {X 0,Y 296.058,Z 776.743,A -85,B 0,C 180,E1 14662.429,E2 14662.429} C_VEL
LIN {X 0,Y 296.292,Z 772.837,A -85,B 0,C 180,E1 14658.711,E2 14658.711} C_VEL
LIN {X 0,Y 297.09,Z 766.881,A -85,B 0,C 180,E1 14654.779,E2 14654.779} C_VEL
LIN {X 0,Y 298.686,Z 758.943,A -85,B 0,C 180,E1 14650.847,E2 14650.847} C_VEL
LIN {X 0,Y 301.255,Z 748.864,A -85,B 0,C 180,E1 14646.942,E2 14646.942} C_VEL
LIN {X 0,Y 304.703,Z 737.116,A -85,B 0,C 180,E1 14643.283,E2 14643.283} C_VEL
LIN {X 0,Y 308.962,Z 723.842,A -85,B 0,C 180,E1 14639.892,E2 14639.892} C_VEL
LIN {X 0,Y 313.936,Z 709.114,A -85,B 0,C 180,E1 14636.782,E2 14636.782} C_VEL
LIN {X 0,Y 320.074,Z 691.451,A -85,B 0,C 180,E1 14633.701,E2 14633.701} C_VEL
LIN {X 0,Y 326.902,Z 672.158,A -85,B 0,C 180,E1 14630.943,E2 14630.943} C_VEL
LIN {X 0,Y 334.096,Z 652.043,A -85,B 0,C 180,E1 14628.592,E2 14628.592} C_VEL
LIN {X 0,Y 341.77,Z 630.618,A -85,B 0,C 180,E1 14626.566,E2 14626.566} C_VEL
LIN {X 0,Y 349.239,Z 609.57,A -85,B 0,C 180,E1 14624.995,E2 14624.995} C_VEL
LIN {X 0,Y 356.52,Z 588.153,A -85,B 0,C 180,E1 14623.765,E2 14623.765} C_VEL
LIN {X 0,Y 362.999,Z 567.158,A -85,B 0,C 180,E1 14622.848,E2 14622.848} C_VEL
LIN {X 0,Y 356.075,Z 588.45,A -85,B 0,C 180,E1 14621.828,E2 14621.828} C_VEL
LIN {X 0,Y 348.708,Z 608.687,A -85,B 0,C 180,E1 14620.499,E2 14620.499} C_VEL
LIN {X 0,Y 340.907,Z 628.961,A -85,B 0,C 180,E1 14618.768,E2 14618.768} C_VEL
LIN {X 0,Y 333.005,Z 649.1,A -85,B 0,C 180,E1 14616.584,E2 14616.584} C_VEL
LIN {X 0,Y 325.721,Z 667.773,A -85,B 0,C 180,E1 14614.07,E2 14614.07} C_VEL
LIN {X 0,Y 319.256,Z 684.33,A -85,B 0,C 180,E1 14611.324,E2 14611.324} C_VEL
LIN {X 0,Y 313.526,Z 699.018,A -85,B 0,C 180,E1 14608.333,E2 14608.333} C_VEL
LIN {X 0,Y 308.596,Z 711.853,A -85,B 0,C 180,E1 14605.115,E2 14605.115} C_VEL
LIN {X 0,Y 304.585,Z 722.584,A -85,B 0,C 180,E1 14601.773,E2 14601.773} C_VEL
LIN {X 0,Y 301.485,Z 731.267,A -85,B 0,C 180,E1 14598.364,E2 14598.364} C_VEL
LIN {X 0,Y 299.226,Z 738.076,A -85,B 0,C 180,E1 14594.909,E2 14594.909} C_VEL
LIN {X 0,Y 297.712,Z 743.131,A -85,B 0,C 180,E1 14591.428,E2 14591.428} C_VEL
LIN {X 0,Y 296.799,Z 746.534,A -85,B 0,C 180,E1 14587.924,E2 14587.924} C_VEL
LIN {X 0,Y 296.337,Z 748.357,A -85,B 0,C 180,E1 14584.256,E2 14584.256} C_VEL
LIN {X 0,Y 296.181,Z 748.441,A -85,B 0,C 180,E1 14580.773,E2 14580.773} C_VEL
LIN {X 0,Y 296.143,Z 746.897,A -85,B 0,C 180,E1 14577.29,E2 14577.29} C_VEL
LIN {X 0,Y 296.246,Z 743.918,A -85,B 0,C 180,E1 14573.994,E2 14573.994} C_VEL
LIN {X 0,Y 296.583,Z 739.38,A -85,B 0,C 180,E1 14570.687,E2 14570.687} C_VEL
LIN {X 0,Y 297.345,Z 732.714,A -85,B 0,C 180,E1 14567.177,E2 14567.177} C_VEL
LIN {X 0,Y 298.573,Z 724.542,A -85,B 0,C 180,E1 14563.861,E2 14563.861} C_VEL
LIN {X 0,Y 300.398,Z 714.286,A -85,B 0,C 180,E1 14560.558,E2 14560.558} C_VEL
LIN {X 0,Y 302.724,Z 702.453,A -85,B 0,C 180,E1 14557.471,E2 14557.471} C_VEL
LIN {X 0,Y 305.487,Z 689.043,A -85,B 0,C 180,E1 14554.605,E2 14554.605} C_VEL
LIN {X 0,Y 308.576,Z 674.094,A -85,B 0,C 180,E1 14551.976,E2 14551.976} C_VEL
LIN {X 0,Y 311.911,Z 657.424,A -85,B 0,C 180,E1 14549.569,E2 14549.569} C_VEL
LIN {X 0,Y 315.11,Z 640.48,A -85,B 0,C 180,E1 14547.571,E2 14547.571} C_VEL
LIN {X 0,Y 318.315,Z 621.836,A -85,B 0,C 180,E1 14545.787,E2 14545.787} C_VEL
LIN {X 0,Y 321.259,Z 602.305,A -85,B 0,C 180,E1 14544.309,E2 14544.309} C_VEL
LIN {X 0,Y 323.833,Z 581.753,A -85,B 0,C 180,E1 14543.132,E2 14543.132} C_VEL
LIN {X 0,Y 325.84,Z 561.087,A -85,B 0,C 180,E1 14542.287,E2 14542.287} C_VEL
LIN {X 0,Y 338.284,Z 387.696,A -85,B 0,C 180,E1 14537.289,E2 14537.289} C_VEL
LIN {X 0,Y 337.288,Z 380.441,A -85,B 0,C 180,E1 14536.887,E2 14536.887} C_VEL
LIN {X 0,Y 324.016,Z 355.169,A -85,B 0,C 180,E1 14534.066,E2 14534.066} C_VEL
LIN {X 0,Y 314.242,Z 337.598,A -85,B 0,C 180,E1 14531.806,E2 14531.806} C_VEL
LIN {X 0,Y 307.561,Z 321.152,A -85,B 0,C 180,E1 14527.912,E2 14527.912} C_VEL
LIN {X 0,Y 301.696,Z 307.291,A -85,B 0,C 180,E1 14524.293,E2 14524.293} C_VEL
LIN {X 0,Y 298.35,Z 299.669,A -85,B 0,C 180,E1 14522.087,E2 14522.087} C_VEL
LIN {X 0,Y 298.344,Z 299.647,A -85,B 0,C 180,E1 14521.651,E2 14521.651} C_VEL
LIN {X 0,Y 299.473,Z 302.618,A -85,B 0,C 180,E1 14520.9,E2 14520.9} C_VEL
LIN {X 0,Y 300.763,Z 304.67,A -85,B 0,C 180,E1 14520.354,E2 14520.354} C_VEL
LIN {X 0,Y 307.285,Z 317.966,A -85,B 0,C 180,E1 14517.311,E2 14517.311} C_VEL
LIN {X 0,Y 313.789,Z 332.45,A -85,B 0,C 180,E1 14514.311,E2 14514.311} C_VEL
LIN {X 0,Y 320.234,Z 349.04,A -85,B 0,C 180,E1 14511.236,E2 14511.236} C_VEL
LIN {X 0,Y 325.746,Z 365.749,A -85,B 0,C 180,E1 14508.432,E2 14508.432} C_VEL
LIN {X 0,Y 326.196,Z 367.588,A -85,B 0,C 180,E1 14508.153,E2 14508.153} C_VEL
LIN {X 0,Y 322.078,Z 408.691,A -85,B 0,C 180,E1 14503.832,E2 14503.832} C_VEL
LIN {X 0,Y 318.024,Z 450.872,A -85,B 0,C 180,E1 14499.411,E2 14499.411} C_VEL
LIN {X 0,Y 315.078,Z 483.048,A -85,B 0,C 180,E1 14496.047,E2 14496.047} C_VEL
LIN {X 0,Y 317.125,Z 505.823,A -85,B 0,C 180,E1 14495.242,E2 14495.242} C_VEL
LIN {X 0,Y 313.15,Z 627.003,A -85,B 0,C 180,E1 14492.427,E2 14492.427} C_VEL
LIN {X 0,Y 312.156,Z 643.081,A -85,B 0,C 180,E1 14491.721,E2 14491.721} C_VEL
LIN {X 0,Y 310.63,Z 659.442,A -85,B 0,C 180,E1 14490.647,E2 14490.647} C_VEL
LIN {X 0,Y 308.843,Z 673.77,A -85,B 0,C 180,E1 14489.353,E2 14489.353} C_VEL
LIN {X 0,Y 306.706,Z 688.146,A -85,B 0,C 180,E1 14487.667,E2 14487.667} C_VEL
LIN {X 0,Y 305.895,Z 693.038,A -85,B 0,C 180,E1 14486.982,E2 14486.982} C_VEL
LIN {X 0,Y 303.942,Z 699.059,A -85,B 0,C 180,E1 14486.136,E2 14486.136} C_VEL
LIN {X 0,Y 297.366,Z 710.104,A -85,B 0,C 180,E1 14484.428,E2 14484.428} C_VEL
LIN {X 0,Y 294.321,Z 715.969,A -85,B 0,C 180,E1 14483.271,E2 14483.271} C_VEL
LIN {X 0,Y 293.713,Z 718.085,A -85,B 0,C 180,E1 14482.784,E2 14482.784} C_VEL
LIN {X 0,Y 291.804,Z 727.607,A -85,B 0,C 180,E1 14480.137,E2 14480.137} C_VEL
LIN {X 0,Y 290.267,Z 735.655,A -85,B 0,C 180,E1 14477.267,E2 14477.267} C_VEL
LIN {X 0,Y 289.154,Z 742.088,A -85,B 0,C 180,E1 14474.149,E2 14474.149} C_VEL
LIN {X 0,Y 288.521,Z 746.641,A -85,B 0,C 180,E1 14470.991,E2 14470.991} C_VEL
LIN {X 0,Y 288.245,Z 749.351,A -85,B 0,C 180,E1 14467.787,E2 14467.787} C_VEL
LIN {X 0,Y 288.194,Z 750.361,A -85,B 0,C 180,E1 14464.522,E2 14464.522} C_VEL
LIN {X 0,Y 288.325,Z 749.547,A -85,B 0,C 180,E1 14461.327,E2 14461.327} C_VEL
LIN {X 0,Y 288.758,Z 746.923,A -85,B 0,C 180,E1 14458.012,E2 14458.012} C_VEL
LIN {X 0,Y 289.613,Z 742.414,A -85,B 0,C 180,E1 14454.795,E2 14454.795} C_VEL
LIN {X 0,Y 290.942,Z 736.368,A -85,B 0,C 180,E1 14451.79,E2 14451.79} C_VEL
LIN {X 0,Y 292.684,Z 728.836,A -85,B 0,C 180,E1 14449.015,E2 14449.015} C_VEL
LIN {X 0,Y 294.971,Z 719.136,A -85,B 0,C 180,E1 14446.255,E2 14446.255} C_VEL
LIN {X 0,Y 297.299,Z 708.873,A -85,B 0,C 180,E1 14443.973,E2 14443.973} C_VEL
LIN {X 0,Y 299.864,Z 696.725,A -85,B 0,C 180,E1 14441.827,E2 14441.827} C_VEL
LIN {X 0,Y 302.288,Z 683.918,A -85,B 0,C 180,E1 14440.041,E2 14440.041} C_VEL
LIN {X 0,Y 304.649,Z 669.337,A -85,B 0,C 180,E1 14438.466,E2 14438.466} C_VEL
LIN {X 0,Y 306.552,Z 654.73,A -85,B 0,C 180,E1 14437.27,E2 14437.27} C_VEL
LIN {X 0,Y 308.074,Z 638.124,A -85,B 0,C 180,E1 14436.307,E2 14436.307} C_VEL
LIN {X 0,Y 308.979,Z 621.885,A -85,B 0,C 180,E1 14435.716,E2 14435.716} C_VEL
LIN {X 0,Y 313.276,Z 504.516,A -85,B 0,C 180,E1 14432.924,E2 14432.924} C_VEL
LIN {X 0,Y 311.269,Z 483.706,A -85,B 0,C 180,E1 14432.007,E2 14432.007} C_VEL
LIN {X 0,Y 315.775,Z 440.448,A -85,B 0,C 180,E1 14427.434,E2 14427.434} C_VEL
LIN {X 0,Y 320.259,Z 399.816,A -85,B 0,C 180,E1 14423.165,E2 14423.165} C_VEL
LIN {X 0,Y 323.216,Z 372.036,A -85,B 0,C 180,E1 14420.272,E2 14420.272} C_VEL
LIN {X 0,Y 318.951,Z 357.97,A -85,B 0,C 180,E1 14417.704,E2 14417.704} C_VEL
LIN {X 0,Y 314.031,Z 344.867,A -85,B 0,C 180,E1 14414.946,E2 14414.946} C_VEL
LIN {X 0,Y 308.721,Z 332.948,A -85,B 0,C 180,E1 14412.029,E2 14412.029} C_VEL
LIN {X 0,Y 304.464,Z 324.564,A -85,B 0,C 180,E1 14409.642,E2 14409.642} C_VEL
LIN {X 0,Y 301.878,Z 319.942,A -85,B 0,C 180,E1 14408.189,E2 14408.189} C_VEL
LIN {X 0,Y 299.851,Z 316.089,A -85,B 0,C 180,E1 14406.895,E2 14406.895} C_VEL
LIN {X 0,Y 297.685,Z 312.569,A -85,B 0,C 180,E1 14405.59,E2 14405.59} C_VEL
LIN {X 0,Y 296.81,Z 311.061,A -85,B 0,C 180,E1 14405.025,E2 14405.025} C_VEL
LIN {X 0,Y 294.525,Z 307.738,A -85,B 0,C 180,E1 14403.6,E2 14403.6} C_VEL
LIN {X 0,Y 293.685,Z 305.893,A -85,B 0,C 180,E1 14402.928,E2 14402.928} C_VEL
LIN {X 0,Y 291.271,Z 303.159,A -85,B 0,C 180,E1 14401.378,E2 14401.378} C_VEL
LIN {X 0,Y 290.382,Z 300.676,A -85,B 0,C 180,E1 14400.297,E2 14400.297} C_VEL
LIN {X 0,Y 290.33,Z 300.314,A -85,B 0,C 180,E1 14398.422,E2 14398.422} C_VEL
LIN {X 0,Y 290.341,Z 300.312,A -85,B 0,C 180,E1 14393.674,E2 14393.674} C_VEL
LIN {X 0,Y 290.352,Z 300.315,A -85,B 0,C 180,E1 14389.083,E2 14389.083} C_VEL
LIN {X 0,Y 290.337,Z 300.31,A -85,B 0,C 180,E1 14384.419,E2 14384.419} C_VEL
LIN {X 0,Y 290.341,Z 300.32,A -85,B 0,C 180,E1 14379.647,E2 14379.647} C_VEL
LIN {X 0,Y 290.353,Z 300.311,A -85,B 0,C 180,E1 14375.159,E2 14375.159} C_VEL
LIN {X 0,Y 290.4,Z 300.603,A -85,B 0,C 180,E1 14372.898,E2 14372.898} C_VEL
LIN {X 0,Y 291.95,Z 304.252,A -85,B 0,C 180,E1 14371.796,E2 14371.796} C_VEL
LIN {X 0,Y 297.957,Z 317.252,A -85,B 0,C 180,E1 14368.208,E2 14368.208} C_VEL
LIN {X 0,Y 300.495,Z 322.749,A -85,B 0,C 180,E1 14366.872,E2 14366.872} C_VEL
LIN {X 0,Y 312.992,Z 342.953,A -85,B 0,C 180,E1 14363.774,E2 14363.774} C_VEL
LIN {X 0,Y 326.944,Z 366.814,A -85,B 0,C 180,E1 14360.64,E2 14360.64} C_VEL
LIN {X 0,Y 337.203,Z 385.814,A -85,B 0,C 180,E1 14358.485,E2 14358.485} C_VEL
LIN {X 0,Y 323.152,Z 576.47,A -85,B 0,C 180,E1 14353.129,E2 14353.129} C_VEL
LIN {X 0,Y 320.716,Z 598.189,A -85,B 0,C 180,E1 14352.206,E2 14352.206} C_VEL
LIN {X 0,Y 317.763,Z 619.003,A -85,B 0,C 180,E1 14350.996,E2 14350.996} C_VEL
LIN {X 0,Y 314.412,Z 638.998,A -85,B 0,C 180,E1 14349.492,E2 14349.492} C_VEL
LIN {X 0,Y 310.637,Z 658.851,A -85,B 0,C 180,E1 14347.609,E2 14347.609} C_VEL
LIN {X 0,Y 306.793,Z 677.253,A -85,B 0,C 180,E1 14345.456,E2 14345.456} C_VEL
LIN {X 0,Y 302.977,Z 694.529,A -85,B 0,C 180,E1 14342.989,E2 14342.989} C_VEL
LIN {X 0,Y 299.277,Z 710.724,A -85,B 0,C 180,E1 14340.183,E2 14340.183} C_VEL
LIN {X 0,Y 295.977,Z 725.269,A -85,B 0,C 180,E1 14337.13,E2 14337.13} C_VEL
LIN {X 0,Y 293.253,Z 737.871,A -85,B 0,C 180,E1 14333.935,E2 14333.935} C_VEL
LIN {X 0,Y 291.083,Z 748.968,A -85,B 0,C 180,E1 14330.507,E2 14330.507} C_VEL
LIN {X 0,Y 289.556,Z 758.27,A -85,B 0,C 180,E1 14326.963,E2 14326.963} C_VEL
LIN {X 0,Y 288.64,Z 765.677,A -85,B 0,C 180,E1 14323.418,E2 14323.418} C_VEL
LIN {X 0,Y 288.223,Z 771.51,A -85,B 0,C 180,E1 14319.785,E2 14319.785} C_VEL
LIN {X 0,Y 288.147,Z 775.657,A -85,B 0,C 180,E1 14316.173,E2 14316.173} C_VEL
LIN {X 0,Y 288.179,Z 777.998,A -85,B 0,C 180,E1 14312.782,E2 14312.782} C_VEL
LIN {X 0,Y 288.182,Z 778.943,A -85,B 0,C 180,E1 14309.203,E2 14309.203} C_VEL
LIN {X 0,Y 288.097,Z 778.471,A -85,B 0,C 180,E1 14305.818,E2 14305.818} C_VEL
LIN {X 0,Y 288.066,Z 776.393,A -85,B 0,C 180,E1 14302.218,E2 14302.218} C_VEL
LIN {X 0,Y 288.327,Z 772.596,A -85,B 0,C 180,E1 14298.395,E2 14298.395} C_VEL
LIN {X 0,Y 289.217,Z 766.77,A -85,B 0,C 180,E1 14294.354,E2 14294.354} C_VEL
LIN {X 0,Y 290.858,Z 759.44,A -85,B 0,C 180,E1 14290.52,E2 14290.52} C_VEL
LIN {X 0,Y 293.432,Z 750.237,A -85,B 0,C 180,E1 14286.715,E2 14286.715} C_VEL
LIN {X 0,Y 297.038,Z 738.999,A -85,B 0,C 180,E1 14282.97,E2 14282.97} C_VEL
LIN {X 0,Y 301.763,Z 725.517,A -85,B 0,C 180,E1 14279.317,E2 14279.317} C_VEL
LIN {X 0,Y 307.353,Z 710.484,A -85,B 0,C 180,E1 14275.974,E2 14275.974} C_VEL
LIN {X 0,Y 313.874,Z 693.503,A -85,B 0,C 180,E1 14272.866,E2 14272.866} C_VEL
LIN {X 0,Y 321.336,Z 674.56,A -85,B 0,C 180,E1 14270.017,E2 14270.017} C_VEL
LIN {X 0,Y 329.771,Z 653.621,A -85,B 0,C 180,E1 14267.456,E2 14267.456} C_VEL
LIN {X 0,Y 338.598,Z 632.089,A -85,B 0,C 180,E1 14265.346,E2 14265.346} C_VEL
LIN {X 0,Y 346.932,Z 611.698,A -85,B 0,C 180,E1 14263.783,E2 14263.783} C_VEL
LIN {X 0,Y 353.303,Z 595.395,A -85,B 0,C 180,E1 14262.781,E2 14262.781} C_VEL
LIN {X 0,Y 345.191,Z 614.593,A -85,B 0,C 180,E1 14261.441,E2 14261.441} C_VEL
LIN {X 0,Y 336.339,Z 634.602,A -85,B 0,C 180,E1 14259.617,E2 14259.617} C_VEL
LIN {X 0,Y 327.74,Z 653.944,A -85,B 0,C 180,E1 14257.38,E2 14257.38} C_VEL
LIN {X 0,Y 319.55,Z 672.365,A -85,B 0,C 180,E1 14254.713,E2 14254.713} C_VEL
LIN {X 0,Y 312.175,Z 689.25,A -85,B 0,C 180,E1 14251.686,E2 14251.686} C_VEL
LIN {X 0,Y 306.281,Z 702.933,A -85,B 0,C 180,E1 14248.677,E2 14248.677} C_VEL
LIN {X 0,Y 301.089,Z 715.166,A -85,B 0,C 180,E1 14245.364,E2 14245.364} C_VEL
LIN {X 0,Y 296.9,Z 725.271,A -85,B 0,C 180,E1 14241.95,E2 14241.95} C_VEL
LIN {X 0,Y 293.669,Z 733.454,A -85,B 0,C 180,E1 14238.459,E2 14238.459} C_VEL
LIN {X 0,Y 291.208,Z 740.129,A -85,B 0,C 180,E1 14234.718,E2 14234.718} C_VEL
LIN {X 0,Y 289.609,Z 744.92,A -85,B 0,C 180,E1 14230.945,E2 14230.945} C_VEL
LIN {X 0,Y 288.741,Z 747.807,A -85,B 0,C 180,E1 14227.361,E2 14227.361} C_VEL
LIN {X 0,Y 288.328,Z 749.088,A -85,B 0,C 180,E1 14223.777,E2 14223.777} C_VEL
LIN {X 0,Y 288.179,Z 748.739,A -85,B 0,C 180,E1 14220.198,E2 14220.198} C_VEL
LIN {X 0,Y 288.157,Z 746.816,A -85,B 0,C 180,E1 14216.695,E2 14216.695} C_VEL
LIN {X 0,Y 288.3,Z 743.34,A -85,B 0,C 180,E1 14213.227,E2 14213.227} C_VEL
LIN {X 0,Y 288.728,Z 738.333,A -85,B 0,C 180,E1 14209.827,E2 14209.827} C_VEL
LIN {X 0,Y 289.635,Z 731.172,A -85,B 0,C 180,E1 14206.219,E2 14206.219} C_VEL
LIN {X 0,Y 291.102,Z 722.203,A -85,B 0,C 180,E1 14202.723,E2 14202.723} C_VEL
LIN {X 0,Y 293.114,Z 711.618,A -85,B 0,C 180,E1 14199.429,E2 14199.429} C_VEL
LIN {X 0,Y 295.699,Z 699.133,A -85,B 0,C 180,E1 14196.272,E2 14196.272} C_VEL
LIN {X 0,Y 298.744,Z 684.919,A -85,B 0,C 180,E1 14193.334,E2 14193.334} C_VEL
LIN {X 0,Y 302.094,Z 669.098,A -85,B 0,C 180,E1 14190.669,E2 14190.669} C_VEL
LIN {X 0,Y 305.413,Z 652.778,A -85,B 0,C 180,E1 14188.411,E2 14188.411} C_VEL
LIN {X 0,Y 308.822,Z 634.784,A -85,B 0,C 180,E1 14186.382,E2 14186.382} C_VEL
LIN {X 0,Y 312.045,Z 615.813,A -85,B 0,C 180,E1 14184.664,E2 14184.664} C_VEL
LIN {X 0,Y 314.995,Z 595.834,A -85,B 0,C 180,E1 14183.248,E2 14183.248} C_VEL
LIN {X 0,Y 317.501,Z 575.057,A -85,B 0,C 180,E1 14182.142,E2 14182.142} C_VEL
LIN {X 0,Y 319.444,Z 553.628,A -85,B 0,C 180,E1 14181.351,E2 14181.351} C_VEL
LIN {X 0,Y 331.795,Z 388.835,A -85,B 0,C 180,E1 14176.496,E2 14176.496} C_VEL
LIN {X 0,Y 331.062,Z 383.919,A -85,B 0,C 180,E1 14176.207,E2 14176.207} C_VEL
LIN {X 0,Y 317.662,Z 358.305,A -85,B 0,C 180,E1 14173.267,E2 14173.267} C_VEL
LIN {X 0,Y 305.918,Z 337.309,A -85,B 0,C 180,E1 14170.439,E2 14170.439} C_VEL
LIN {X 0,Y 299.661,Z 322.098,A -85,B 0,C 180,E1 14166.676,E2 14166.676} C_VEL
LIN {X 0,Y 293.724,Z 308.207,A -85,B 0,C 180,E1 14162.887,E2 14162.887} C_VEL
LIN {X 0,Y 292.649,Z 305.817,A -85,B 0,C 180,E1 14162.078,E2 14162.078} C_VEL
LIN {X 0,Y 292.995,Z 305.922,A -85,B 0,C 180,E1 14161.817,E2 14161.817} C_VEL
LIN {X 0,Y 299.337,Z 318.491,A -85,B 0,C 180,E1 14158.752,E2 14158.752} C_VEL
LIN {X 0,Y 305.719,Z 332.398,A -85,B 0,C 180,E1 14155.705,E2 14155.705} C_VEL
LIN {X 0,Y 312.314,Z 348.839,A -85,B 0,C 180,E1 14152.485,E2 14152.485} C_VEL
LIN {X 0,Y 317.97,Z 365.473,A -85,B 0,C 180,E1 14149.568,E2 14149.568} C_VEL
LIN {X 0,Y 319.369,Z 370.759,A -85,B 0,C 180,E1 14148.719,E2 14148.719} C_VEL
LIN {X 0,Y 315.086,Z 412.181,A -85,B 0,C 180,E1 14144.332,E2 14144.332} C_VEL
LIN {X 0,Y 310.52,Z 457.184,A -85,B 0,C 180,E1 14139.547,E2 14139.547} C_VEL
LIN {X 0,Y 308.06,Z 483.467,A -85,B 0,C 180,E1 14136.774,E2 14136.774} C_VEL
LIN {X 0,Y 310.091,Z 506.691,A -85,B 0,C 180,E1 14135.93,E2 14135.93} C_VEL
LIN {X 0,Y 305.942,Z 627.479,A -85,B 0,C 180,E1 14133.064,E2 14133.064} C_VEL
LIN {X 0,Y 304.89,Z 643.68,A -85,B 0,C 180,E1 14132.334,E2 14132.334} C_VEL
LIN {X 0,Y 303.423,Z 658.854,A -85,B 0,C 180,E1 14131.324,E2 14131.324} C_VEL
LIN {X 0,Y 301.562,Z 673.458,A -85,B 0,C 180,E1 14130.002,E2 14130.002} C_VEL
LIN {X 0,Y 299.322,Z 687.963,A -85,B 0,C 180,E1 14128.279,E2 14128.279} C_VEL
LIN {X 0,Y 297.06,Z 700.729,A -85,B 0,C 180,E1 14126.336,E2 14126.336} C_VEL
LIN {X 0,Y 294.728,Z 712.976,A -85,B 0,C 180,E1 14123.965,E2 14123.965} C_VEL
LIN {X 0,Y 293.713,Z 718.085,A -85,B 0,C 180,E1 14122.784,E2 14122.784} C_VEL
LIN {X 0,Y 291.83,Z 722.819,A -85,B 0,C 180,E1 14121.635,E2 14121.635} C_VEL
LIN {X 0,Y 285.957,Z 730.647,A -85,B 0,C 180,E1 14119.497,E2 14119.497} C_VEL
LIN {X 0,Y 282.972,Z 734.859,A -85,B 0,C 180,E1 14118.03,E2 14118.03} C_VEL
LIN {X 0,Y 282.245,Z 736.774,A -85,B 0,C 180,E1 14117.23,E2 14117.23} C_VEL
LIN {X 0,Y 281.151,Z 742.896,A -85,B 0,C 180,E1 14114.11,E2 14114.11} C_VEL
LIN {X 0,Y 280.543,Z 747.061,A -85,B 0,C 180,E1 14111.078,E2 14111.078} C_VEL
LIN {X 0,Y 280.254,Z 749.76,A -85,B 0,C 180,E1 14107.782,E2 14107.782} C_VEL
LIN {X 0,Y 280.205,Z 750.754,A -85,B 0,C 180,E1 14104.423,E2 14104.423} C_VEL
LIN {X 0,Y 280.346,Z 749.97,A -85,B 0,C 180,E1 14101.221,E2 14101.221} C_VEL
LIN {X 0,Y 280.786,Z 747.499,A -85,B 0,C 180,E1 14097.942,E2 14097.942} C_VEL
LIN {X 0,Y 281.65,Z 743.296,A -85,B 0,C 180,E1 14094.738,E2 14094.738} C_VEL
LIN {X 0,Y 283.066,Z 737.211,A -85,B 0,C 180,E1 14091.565,E2 14091.565} C_VEL
LIN {X 0,Y 284.919,Z 729.728,A -85,B 0,C 180,E1 14088.677,E2 14088.677} C_VEL
LIN {X 0,Y 287.365,Z 719.911,A -85,B 0,C 180,E1 14085.789,E2 14085.789} C_VEL
LIN {X 0,Y 289.96,Z 709.115,A -85,B 0,C 180,E1 14083.32,E2 14083.32} C_VEL
LIN {X 0,Y 292.694,Z 696.846,A -85,B 0,C 180,E1 14081.11,E2 14081.11} C_VEL
LIN {X 0,Y 295.237,Z 684.023,A -85,B 0,C 180,E1 14079.295,E2 14079.295} C_VEL
LIN {X 0,Y 297.737,Z 669.235,A -85,B 0,C 180,E1 14077.677,E2 14077.677} C_VEL
LIN {X 0,Y 299.684,Z 654.783,A -85,B 0,C 180,E1 14076.484,E2 14076.484} C_VEL
LIN {X 0,Y 301.286,Z 637.985,A -85,B 0,C 180,E1 14075.502,E2 14075.502} C_VEL
LIN {X 0,Y 302.215,Z 621.596,A -85,B 0,C 180,E1 14074.908,E2 14074.908} C_VEL
LIN {X 0,Y 306.717,Z 505.397,A -85,B 0,C 180,E1 14072.085,E2 14072.085} C_VEL
LIN {X 0,Y 304.744,Z 483.938,A -85,B 0,C 180,E1 14071.098,E2 14071.098} C_VEL
LIN {X 0,Y 309.476,Z 440.771,A -85,B 0,C 180,E1 14066.479,E2 14066.479} C_VEL
LIN {X 0,Y 313.94,Z 402.011,A -85,B 0,C 180,E1 14062.371,E2 14062.371} C_VEL
LIN {X 0,Y 316.94,Z 375.31,A -85,B 0,C 180,E1 14059.537,E2 14059.537} C_VEL
LIN {X 0,Y 312.814,Z 361.491,A -85,B 0,C 180,E1 14056.911,E2 14056.911} C_VEL
LIN {X 0,Y 308.061,Z 348.584,A -85,B 0,C 180,E1 14054.089,E2 14054.089} C_VEL
LIN {X 0,Y 302.482,Z 336.042,A -85,B 0,C 180,E1 14050.861,E2 14050.861} C_VEL
LIN {X 0,Y 297.914,Z 327.046,A -85,B 0,C 180,E1 14048.104,E2 14048.104} C_VEL
LIN {X 0,Y 295.304,Z 322.305,A -85,B 0,C 180,E1 14046.416,E2 14046.416} C_VEL
LIN {X 0,Y 292.649,Z 317.725,A -85,B 0,C 180,E1 14044.704,E2 14044.704} C_VEL
LIN {X 0,Y 290.362,Z 314.198,A -85,B 0,C 180,E1 14043.159,E2 14043.159} C_VEL
LIN {X 0,Y 289.655,Z 312.683,A -85,B 0,C 180,E1 14042.573,E2 14042.573} C_VEL
LIN {X 0,Y 287.148,Z 309.419,A -85,B 0,C 180,E1 14040.799,E2 14040.799} C_VEL
LIN {X 0,Y 285.949,Z 307.02,A -85,B 0,C 180,E1 14039.707,E2 14039.707} C_VEL
LIN {X 0,Y 283.212,Z 303.942,A -85,B 0,C 180,E1 14037.512,E2 14037.512} C_VEL
LIN {X 0,Y 282.445,Z 301.673,A -85,B 0,C 180,E1 14036.246,E2 14036.246} C_VEL
LIN {X 0,Y 282.401,Z 301.3,A -85,B 0,C 180,E1 14033.699,E2 14033.699} C_VEL
LIN {X 0,Y 282.411,Z 301.306,A -85,B 0,C 180,E1 14028.979,E2 14028.979} C_VEL
LIN {X 0,Y 282.397,Z 301.299,A -85,B 0,C 180,E1 14024.365,E2 14024.365} C_VEL
LIN {X 0,Y 282.401,Z 301.309,A -85,B 0,C 180,E1 14019.698,E2 14019.698} C_VEL
LIN {X 0,Y 282.414,Z 301.3,A -85,B 0,C 180,E1 14015.084,E2 14015.084} C_VEL
LIN {X 0,Y 282.492,Z 301.857,A -85,B 0,C 180,E1 14014.418,E2 14014.418} C_VEL
LIN {X 0,Y 283.883,Z 305.035,A -85,B 0,C 180,E1 14013.43,E2 14013.43} C_VEL
LIN {X 0,Y 288.805,Z 315.63,A -85,B 0,C 180,E1 14010.326,E2 14010.326} C_VEL
LIN {X 0,Y 292.298,Z 322.994,A -85,B 0,C 180,E1 14008.385,E2 14008.385} C_VEL
LIN {X 0,Y 305.566,Z 344.296,A -85,B 0,C 180,E1 14004.953,E2 14004.953} C_VEL
LIN {X 0,Y 319.74,Z 368.482,A -85,B 0,C 180,E1 14001.631,E2 14001.631} C_VEL
LIN {X 0,Y 330.685,Z 388.558,A -85,B 0,C 180,E1 13999.258,E2 13999.258} C_VEL
LIN {X 0,Y 316.201,Z 576.44,A -85,B 0,C 180,E1 13993.839,E2 13993.839} C_VEL
LIN {X 0,Y 313.756,Z 597.587,A -85,B 0,C 180,E1 13992.925,E2 13992.925} C_VEL
LIN {X 0,Y 310.649,Z 618.855,A -85,B 0,C 180,E1 13991.666,E2 13991.666} C_VEL
LIN {X 0,Y 307.081,Z 639.415,A -85,B 0,C 180,E1 13990.079,E2 13990.079} C_VEL
LIN {X 0,Y 303.249,Z 658.915,A -85,B 0,C 180,E1 13988.183,E2 13988.183} C_VEL
LIN {X 0,Y 299.33,Z 677.098,A -85,B 0,C 180,E1 13986.005,E2 13986.005} C_VEL
LIN {X 0,Y 295.394,Z 694.354,A -85,B 0,C 180,E1 13983.483,E2 13983.483} C_VEL
LIN {X 0,Y 291.695,Z 710.039,A -85,B 0,C 180,E1 13980.71,E2 13980.71} C_VEL
LIN {X 0,Y 288.371,Z 724.231,A -85,B 0,C 180,E1 13977.682,E2 13977.682} C_VEL
LIN {X 0,Y 285.363,Z 737.674,A -85,B 0,C 180,E1 13974.199,E2 13974.199} C_VEL
LIN {X 0,Y 283.102,Z 748.923,A -85,B 0,C 180,E1 13970.623,E2 13970.623} C_VEL
LIN {X 0,Y 281.531,Z 758.289,A -85,B 0,C 180,E1 13966.929,E2 13966.929} C_VEL
LIN {X 0,Y 280.602,Z 765.79,A -85,B 0,C 180,E1 13963.18,E2 13963.18} C_VEL
LIN {X 0,Y 280.218,Z 771.466,A -85,B 0,C 180,E1 13959.445,E2 13959.445} C_VEL
LIN {X 0,Y 280.161,Z 775.729,A -85,B 0,C 180,E1 13955.527,E2 13955.527} C_VEL
LIN {X 0,Y 280.205,Z 777.704,A -85,B 0,C 180,E1 13952.247,E2 13952.247} C_VEL
LIN {X 0,Y 280.19,Z 778.447,A -85,B 0,C 180,E1 13948.771,E2 13948.771} C_VEL
LIN {X 0,Y 280.083,Z 777.8,A -85,B 0,C 180,E1 13945.083,E2 13945.083} C_VEL
LIN {X 0,Y 280.094,Z 775.614,A -85,B 0,C 180,E1 13941.375,E2 13941.375} C_VEL
LIN {X 0,Y 280.465,Z 771.646,A -85,B 0,C 180,E1 13937.438,E2 13937.438} C_VEL
LIN {X 0,Y 281.59,Z 765.677,A -85,B 0,C 180,E1 13933.283,E2 13933.283} C_VEL
LIN {X 0,Y 283.72,Z 757.558,A -85,B 0,C 180,E1 13929.048,E2 13929.048} C_VEL
LIN {X 0,Y 287.047,Z 747.253,A -85,B 0,C 180,E1 13924.85,E2 13924.85} C_VEL
LIN {X 0,Y 291.557,Z 734.966,A -85,B 0,C 180,E1 13920.856,E2 13920.856} C_VEL
LIN {X 0,Y 297.072,Z 721.083,A -85,B 0,C 180,E1 13917.186,E2 13917.186} C_VEL
LIN {X 0,Y 303.712,Z 705.238,A -85,B 0,C 180,E1 13913.761,E2 13913.761} C_VEL
LIN {X 0,Y 311.353,Z 687.627,A -85,B 0,C 180,E1 13910.635,E2 13910.635} C_VEL
LIN {X 0,Y 320.1,Z 668.143,A -85,B 0,C 180,E1 13907.81,E2 13907.81} C_VEL
LIN {X 0,Y 329.945,Z 646.738,A -85,B 0,C 180,E1 13905.326,E2 13905.326} C_VEL
LIN {X 0,Y 339.525,Z 626.321,A -85,B 0,C 180,E1 13903.453,E2 13903.453} C_VEL
LIN {X 0,Y 343.988,Z 616.74,A -85,B 0,C 180,E1 13902.714,E2 13902.714} C_VEL
LIN {X 0,Y 334.182,Z 636.164,A -85,B 0,C 180,E1 13900.937,E2 13900.937} C_VEL
LIN {X 0,Y 324.551,Z 655.099,A -85,B 0,C 180,E1 13898.71,E2 13898.71} C_VEL
LIN {X 0,Y 315.626,Z 672.769,A -85,B 0,C 180,E1 13896.101,E2 13896.101} C_VEL
LIN {X 0,Y 307.533,Z 689.18,A -85,B 0,C 180,E1 13893.106,E2 13893.106} C_VEL
LIN {X 0,Y 300.683,Z 703.374,A -85,B 0,C 180,E1 13889.92,E2 13889.92} C_VEL
LIN {X 0,Y 294.685,Z 716.038,A -85,B 0,C 180,E1 13886.389,E2 13886.389} C_VEL
LIN {X 0,Y 289.864,Z 726.446,A -85,B 0,C 180,E1 13882.726,E2 13882.726} C_VEL
LIN {X 0,Y 286.166,Z 734.798,A -85,B 0,C 180,E1 13878.961,E2 13878.961} C_VEL
LIN {X 0,Y 283.507,Z 741.218,A -85,B 0,C 180,E1 13875.128,E2 13875.128} C_VEL
LIN {X 0,Y 281.765,Z 745.798,A -85,B 0,C 180,E1 13871.254,E2 13871.254} C_VEL
LIN {X 0,Y 280.773,Z 748.591,A -85,B 0,C 180,E1 13867.365,E2 13867.365} C_VEL
LIN {X 0,Y 280.337,Z 749.626,A -85,B 0,C 180,E1 13863.68,E2 13863.68} C_VEL
LIN {X 0,Y 280.187,Z 749.061,A -85,B 0,C 180,E1 13859.999,E2 13859.999} C_VEL
LIN {X 0,Y 280.169,Z 746.862,A -85,B 0,C 180,E1 13856.316,E2 13856.316} C_VEL
LIN {X 0,Y 280.357,Z 742.956,A -85,B 0,C 180,E1 13852.623,E2 13852.623} C_VEL
LIN {X 0,Y 280.912,Z 737.225,A -85,B 0,C 180,E1 13848.918,E2 13848.918} C_VEL
LIN {X 0,Y 281.983,Z 729.517,A -85,B 0,C 180,E1 13845.208,E2 13845.208} C_VEL
LIN {X 0,Y 283.611,Z 720.236,A -85,B 0,C 180,E1 13841.713,E2 13841.713} C_VEL
LIN {X 0,Y 285.77,Z 709.469,A -85,B 0,C 180,E1 13838.445,E2 13838.445} C_VEL
LIN {X 0,Y 288.393,Z 697.285,A -85,B 0,C 180,E1 13835.414,E2 13835.414} C_VEL
LIN {X 0,Y 291.504,Z 683.172,A -85,B 0,C 180,E1 13832.526,E2 13832.526} C_VEL
LIN {X 0,Y 294.929,Z 667.46,A -85,B 0,C 180,E1 13829.884,E2 13829.884} C_VEL
LIN {X 0,Y 298.561,Z 650.003,A -85,B 0,C 180,E1 13827.485,E2 13827.485} C_VEL
LIN {X 0,Y 301.977,Z 632.326,A -85,B 0,C 180,E1 13825.514,E2 13825.514} C_VEL
LIN {X 0,Y 305.283,Z 613.192,A -85,B 0,C 180,E1 13823.799,E2 13823.799} C_VEL
LIN {X 0,Y 308.319,Z 592.759,A -85,B 0,C 180,E1 13822.375,E2 13822.375} C_VEL
LIN {X 0,Y 310.864,Z 571.524,A -85,B 0,C 180,E1 13821.288,E2 13821.288} C_VEL
LIN {X 0,Y 312.978,Z 547.09,A -85,B 0,C 180,E1 13820.428,E2 13820.428} C_VEL
LIN {X 0,Y 325.336,Z 390.045,A -85,B 0,C 180,E1 13815.687,E2 13815.687} C_VEL
LIN {X 0,Y 324.759,Z 387.177,A -85,B 0,C 180,E1 13815.491,E2 13815.491} C_VEL
LIN {X 0,Y 311.766,Z 362.38,A -85,B 0,C 180,E1 13812.557,E2 13812.557} C_VEL
LIN {X 0,Y 299.503,Z 340.601,A -85,B 0,C 180,E1 13809.556,E2 13809.556} C_VEL
LIN {X 0,Y 297.465,Z 336.802,A -85,B 0,C 180,E1 13808.946,E2 13808.946} C_VEL
LIN {X 0,Y 290.856,Z 320.692,A -85,B 0,C 180,E1 13804.754,E2 13804.754} C_VEL
LIN {X 0,Y 287.28,Z 312.589,A -85,B 0,C 180,E1 13802.375,E2 13802.375} C_VEL
LIN {X 0,Y 287.974,Z 312.566,A -85,B 0,C 180,E1 13801.951,E2 13801.951} C_VEL
LIN {X 0,Y 291.896,Z 320.133,A -85,B 0,C 180,E1 13800.009,E2 13800.009} C_VEL
LIN {X 0,Y 298.485,Z 334.191,A -85,B 0,C 180,E1 13796.781,E2 13796.781} C_VEL
LIN {X 0,Y 304.835,Z 349.874,A -85,B 0,C 180,E1 13793.59,E2 13793.59} C_VEL
LIN {X 0,Y 310.826,Z 367.12,A -85,B 0,C 180,E1 13790.439,E2 13790.439} C_VEL
LIN {X 0,Y 312.652,Z 373.507,A -85,B 0,C 180,E1 13789.366,E2 13789.366} C_VEL
LIN {X 0,Y 308.169,Z 414.628,A -85,B 0,C 180,E1 13784.95,E2 13784.95} C_VEL
LIN {X 0,Y 303.645,Z 457.497,A -85,B 0,C 180,E1 13780.34,E2 13780.34} C_VEL
LIN {X 0,Y 301.084,Z 483.752,A -85,B 0,C 180,E1 13777.539,E2 13777.539} C_VEL
LIN {X 0,Y 303.106,Z 507.478,A -85,B 0,C 180,E1 13776.652,E2 13776.652} C_VEL
LIN {X 0,Y 298.757,Z 627.929,A -85,B 0,C 180,E1 13773.726,E2 13773.726} C_VEL
LIN {X 0,Y 297.652,Z 644.202,A -85,B 0,C 180,E1 13772.975,E2 13772.975} C_VEL
LIN {X 0,Y 296.117,Z 659.427,A -85,B 0,C 180,E1 13771.937,E2 13771.937} C_VEL
LIN {X 0,Y 294.181,Z 673.985,A -85,B 0,C 180,E1 13770.586,E2 13770.586} C_VEL
LIN {X 0,Y 291.849,Z 688.476,A -85,B 0,C 180,E1 13768.824,E2 13768.824} C_VEL
LIN {X 0,Y 289.491,Z 701.221,A -85,B 0,C 180,E1 13766.834,E2 13766.834} C_VEL
LIN {X 0,Y 287.056,Z 713.46,A -85,B 0,C 180,E1 13764.405,E2 13764.405} C_VEL
LIN {X 0,Y 284.89,Z 723.782,A -85,B 0,C 180,E1 13761.783,E2 13761.783} C_VEL
LIN {X 0,Y 283.121,Z 732.348,A -85,B 0,C 180,E1 13759.009,E2 13759.009} C_VEL
LIN {X 0,Y 282.245,Z 736.774,A -85,B 0,C 180,E1 13757.23,E2 13757.23} C_VEL
LIN {X 0,Y 280.683,Z 739.906,A -85,B 0,C 180,E1 13755.813,E2 13755.813} C_VEL
LIN {X 0,Y 275.672,Z 744.607,A -85,B 0,C 180,E1 13753.301,E2 13753.301} C_VEL
LIN {X 0,Y 272.862,Z 747.256,A -85,B 0,C 180,E1 13751.36,E2 13751.36} C_VEL
LIN {X 0,Y 272.485,Z 748.065,A -85,B 0,C 180,E1 13750.564,E2 13750.564} C_VEL
LIN {X 0,Y 272.241,Z 750.478,A -85,B 0,C 180,E1 13747.2,E2 13747.2} C_VEL
LIN {X 0,Y 272.224,Z 751.109,A -85,B 0,C 180,E1 13743.851,E2 13743.851} C_VEL
LIN {X 0,Y 272.432,Z 750.061,A -85,B 0,C 180,E1 13740.439,E2 13740.439} C_VEL
LIN {X 0,Y 272.961,Z 747.379,A -85,B 0,C 180,E1 13737.175,E2 13737.175} C_VEL
LIN {X 0,Y 274.037,Z 742.664,A -85,B 0,C 180,E1 13733.742,E2 13733.742} C_VEL
LIN {X 0,Y 275.619,Z 736.449,A -85,B 0,C 180,E1 13730.595,E2 13730.595} C_VEL
LIN {X 0,Y 277.861,Z 727.994,A -85,B 0,C 180,E1 13727.433,E2 13727.433} C_VEL
LIN {X 0,Y 280.299,Z 718.761,A -85,B 0,C 180,E1 13724.781,E2 13724.781} C_VEL
LIN {X 0,Y 283.233,Z 707.063,A -85,B 0,C 180,E1 13722.159,E2 13722.159} C_VEL
LIN {X 0,Y 286.023,Z 694.923,A -85,B 0,C 180,E1 13720.033,E2 13720.033} C_VEL
LIN {X 0,Y 288.739,Z 681.488,A -85,B 0,C 180,E1 13718.185,E2 13718.185} C_VEL
LIN {X 0,Y 291.143,Z 667.519,A -85,B 0,C 180,E1 13716.696,E2 13716.696} C_VEL
LIN {X 0,Y 293.284,Z 651.386,A -85,B 0,C 180,E1 13715.421,E2 13715.421} C_VEL
LIN {X 0,Y 294.752,Z 635.543,A -85,B 0,C 180,E1 13714.551,E2 13714.551} C_VEL
LIN {X 0,Y 295.692,Z 617.171,A -85,B 0,C 180,E1 13713.951,E2 13713.951} C_VEL
LIN {X 0,Y 300.247,Z 506.37,A -85,B 0,C 180,E1 13711.209,E2 13711.209} C_VEL
LIN {X 0,Y 298.26,Z 484.586,A -85,B 0,C 180,E1 13710.189,E2 13710.189} C_VEL
LIN {X 0,Y 303.278,Z 441.118,A -85,B 0,C 180,E1 13705.483,E2 13705.483} C_VEL
LIN {X 0,Y 308.284,Z 400.374,A -85,B 0,C 180,E1 13701.101,E2 13701.101} C_VEL
LIN {X 0,Y 310.833,Z 378.715,A -85,B 0,C 180,E1 13698.765,E2 13698.765} C_VEL
LIN {X 0,Y 306.761,Z 365.002,A -85,B 0,C 180,E1 13696.085,E2 13696.085} C_VEL
LIN {X 0,Y 302.148,Z 352.38,A -85,B 0,C 180,E1 13693.2,E2 13693.2} C_VEL
LIN {X 0,Y 297.407,Z 341.469,A -85,B 0,C 180,E1 13690.265,E2 13690.265} C_VEL
LIN {X 0,Y 292.716,Z 332.185,A -85,B 0,C 180,E1 13687.261,E2 13687.261} C_VEL
LIN {X 0,Y 290.789,Z 328.5,A -85,B 0,C 180,E1 13685.921,E2 13685.921} C_VEL
LIN {X 0,Y 288.17,Z 324.01,A -85,B 0,C 180,E1 13684.179,E2 13684.179} C_VEL
LIN {X 0,Y 285.709,Z 319.489,A -85,B 0,C 180,E1 13682.207,E2 13682.207} C_VEL
LIN {X 0,Y 283.292,Z 316.154,A -85,B 0,C 180,E1 13680.405,E2 13680.405} C_VEL
LIN {X 0,Y 282.211,Z 313.989,A -85,B 0,C 180,E1 13679.392,E2 13679.392} C_VEL
LIN {X 0,Y 279.643,Z 310.853,A -85,B 0,C 180,E1 13677.131,E2 13677.131} C_VEL
LIN {X 0,Y 278.473,Z 308.311,A -85,B 0,C 180,E1 13675.676,E2 13675.676} C_VEL
LIN {X 0,Y 275.202,Z 304.808,A -85,B 0,C 180,E1 13671.855,E2 13671.855} C_VEL
LIN {X 0,Y 274.529,Z 302.767,A -85,B 0,C 180,E1 13669.933,E2 13669.933} C_VEL
LIN {X 0,Y 274.475,Z 302.286,A -85,B 0,C 180,E1 13666.948,E2 13666.948} C_VEL
LIN {X 0,Y 274.458,Z 302.294,A -85,B 0,C 180,E1 13662.181,E2 13662.181} C_VEL
LIN {X 0,Y 274.484,Z 302.316,A -85,B 0,C 180,E1 13657.287,E2 13657.287} C_VEL
LIN {X 0,Y 274.51,Z 302.633,A -85,B 0,C 180,E1 13656.223,E2 13656.223} C_VEL
LIN {X 0,Y 276.194,Z 306.361,A -85,B 0,C 180,E1 13654.941,E2 13654.941} C_VEL
LIN {X 0,Y 282.302,Z 319.458,A -85,B 0,C 180,E1 13650.973,E2 13650.973} C_VEL
LIN {X 0,Y 284.199,Z 323.388,A -85,B 0,C 180,E1 13649.941,E2 13649.941} C_VEL
LIN {X 0,Y 297.646,Z 344.923,A -85,B 0,C 180,E1 13646.282,E2 13646.282} C_VEL
LIN {X 0,Y 311.043,Z 367.574,A -85,B 0,C 180,E1 13642.993,E2 13642.993} C_VEL
LIN {X 0,Y 324.168,Z 391.398,A -85,B 0,C 180,E1 13640.048,E2 13640.048} C_VEL
LIN {X 0,Y 309.274,Z 576.305,A -85,B 0,C 180,E1 13634.573,E2 13634.573} C_VEL
LIN {X 0,Y 306.783,Z 597.161,A -85,B 0,C 180,E1 13633.653,E2 13633.653} C_VEL
LIN {X 0,Y 303.743,Z 617.505,A -85,B 0,C 180,E1 13632.436,E2 13632.436} C_VEL
LIN {X 0,Y 300.178,Z 637.626,A -85,B 0,C 180,E1 13630.878,E2 13630.878} C_VEL
LIN {X 0,Y 296.114,Z 657.791,A -85,B 0,C 180,E1 13628.903,E2 13628.903} C_VEL
LIN {X 0,Y 292.057,Z 676.129,A -85,B 0,C 180,E1 13626.678,E2 13626.678} C_VEL
LIN {X 0,Y 287.979,Z 693.486,A -85,B 0,C 180,E1 13624.103,E2 13624.103} C_VEL
LIN {X 0,Y 284.014,Z 709.769,A -85,B 0,C 180,E1 13621.162,E2 13621.162} C_VEL
LIN {X 0,Y 280.583,Z 723.971,A -85,B 0,C 180,E1 13618.056,E2 13618.056} C_VEL
LIN {X 0,Y 277.481,Z 737.412,A -85,B 0,C 180,E1 13614.478,E2 13614.478} C_VEL
LIN {X 0,Y 275.182,Z 748.503,A -85,B 0,C 180,E1 13610.857,E2 13610.857} C_VEL
LIN {X 0,Y 273.543,Z 758.012,A -85,B 0,C 180,E1 13607,E2 13607} C_VEL
LIN {X 0,Y 272.604,Z 765.487,A -85,B 0,C 180,E1 13603.142,E2 13603.142} C_VEL
LIN {X 0,Y 272.197,Z 772.186,A -85,B 0,C 180,E1 13598.66,E2 13598.66} C_VEL
LIN {X 0,Y 272.163,Z 775.703,A -85,B 0,C 180,E1 13595.267,E2 13595.267} C_VEL
LIN {X 0,Y 272.215,Z 777.363,A -85,B 0,C 180,E1 13592.103,E2 13592.103} C_VEL
LIN {X 0,Y 272.188,Z 777.946,A -85,B 0,C 180,E1 13588.103,E2 13588.103} C_VEL
LIN {X 0,Y 272.08,Z 777.126,A -85,B 0,C 180,E1 13584.303,E2 13584.303} C_VEL
LIN {X 0,Y 272.127,Z 774.839,A -85,B 0,C 180,E1 13580.481,E2 13580.481} C_VEL
LIN {X 0,Y 272.675,Z 770.631,A -85,B 0,C 180,E1 13576.338,E2 13576.338} C_VEL
LIN {X 0,Y 274.046,Z 764.625,A -85,B 0,C 180,E1 13572.151,E2 13572.151} C_VEL
LIN {X 0,Y 276.479,Z 756.619,A -85,B 0,C 180,E1 13567.905,E2 13567.905} C_VEL
LIN {X 0,Y 280.129,Z 746.625,A -85,B 0,C 180,E1 13563.729,E2 13563.729} C_VEL
LIN {X 0,Y 285.114,Z 734.504,A -85,B 0,C 180,E1 13559.667,E2 13559.667} C_VEL
LIN {X 0,Y 291.544,Z 720.009,A -85,B 0,C 180,E1 13555.742,E2 13555.742} C_VEL
LIN {X 0,Y 298.948,Z 704.206,A -85,B 0,C 180,E1 13552.259,E2 13552.259} C_VEL
LIN {X 0,Y 307.58,Z 686.563,A -85,B 0,C 180,E1 13549.077,E2 13549.077} C_VEL
LIN {X 0,Y 317.689,Z 666.722,A -85,B 0,C 180,E1 13546.177,E2 13546.177} C_VEL
LIN {X 0,Y 328.403,Z 646.394,A -85,B 0,C 180,E1 13543.814,E2 13543.814} C_VEL
LIN {X 0,Y 334.839,Z 634.376,A -85,B 0,C 180,E1 13542.648,E2 13542.648} C_VEL
LIN {X 0,Y 323.905,Z 653.14,A -85,B 0,C 180,E1 13540.525,E2 13540.525} C_VEL
LIN {X 0,Y 313.697,Z 670.924,A -85,B 0,C 180,E1 13537.963,E2 13537.963} C_VEL
LIN {X 0,Y 304.158,Z 687.883,A -85,B 0,C 180,E1 13534.888,E2 13534.888} C_VEL
LIN {X 0,Y 296.096,Z 702.657,A -85,B 0,C 180,E1 13531.56,E2 13531.56} C_VEL
LIN {X 0,Y 289.375,Z 715.279,A -85,B 0,C 180,E1 13528.028,E2 13528.028} C_VEL
LIN {X 0,Y 283.92,Z 725.821,A -85,B 0,C 180,E1 13524.332,E2 13524.332} C_VEL
LIN {X 0,Y 279.598,Z 734.456,A -85,B 0,C 180,E1 13520.454,E2 13520.454} C_VEL
LIN {X 0,Y 276.353,Z 741.257,A -85,B 0,C 180,E1 13516.391,E2 13516.391} C_VEL
LIN {X 0,Y 274.263,Z 745.975,A -85,B 0,C 180,E1 13512.42,E2 13512.42} C_VEL
LIN {X 0,Y 273.02,Z 748.937,A -85,B 0,C 180,E1 13508.423,E2 13508.423} C_VEL
LIN {X 0,Y 272.416,Z 750.157,A -85,B 0,C 180,E1 13504.42,E2 13504.42} C_VEL
LIN {X 0,Y 272.211,Z 749.687,A -85,B 0,C 180,E1 13500.631,E2 13500.631} C_VEL
LIN {X 0,Y 272.167,Z 747.573,A -85,B 0,C 180,E1 13496.84,E2 13496.84} C_VEL
LIN {X 0,Y 272.307,Z 744.018,A -85,B 0,C 180,E1 13493.251,E2 13493.251} C_VEL
LIN {X 0,Y 272.76,Z 738.867,A -85,B 0,C 180,E1 13489.652,E2 13489.652} C_VEL
LIN {X 0,Y 273.669,Z 731.999,A -85,B 0,C 180,E1 13486.046,E2 13486.046} C_VEL
LIN {X 0,Y 275.176,Z 723.231,A -85,B 0,C 180,E1 13482.446,E2 13482.446} C_VEL
LIN {X 0,Y 277.223,Z 713.013,A -85,B 0,C 180,E1 13479.079,E2 13479.079} C_VEL
LIN {X 0,Y 279.753,Z 701.429,A -85,B 0,C 180,E1 13475.955,E2 13475.955} C_VEL
LIN {X 0,Y 282.902,Z 687.553,A -85,B 0,C 180,E1 13472.875,E2 13472.875} C_VEL
LIN {X 0,Y 286.29,Z 672.63,A -85,B 0,C 180,E1 13470.153,E2 13470.153} C_VEL
LIN {X 0,Y 289.906,Z 656.104,A -85,B 0,C 180,E1 13467.673,E2 13467.673} C_VEL
LIN {X 0,Y 293.625,Z 637.936,A -85,B 0,C 180,E1 13465.46,E2 13465.46} C_VEL
LIN {X 0,Y 297.011,Z 619.609,A -85,B 0,C 180,E1 13463.665,E2 13463.665} C_VEL
LIN {X 0,Y 300.092,Z 600.611,A -85,B 0,C 180,E1 13462.188,E2 13462.188} C_VEL
LIN {X 0,Y 302.879,Z 580.053,A -85,B 0,C 180,E1 13460.967,E2 13460.967} C_VEL
LIN {X 0,Y 305.192,Z 558.06,A -85,B 0,C 180,E1 13460.041,E2 13460.041} C_VEL
LIN {X 0,Y 318.928,Z 391.443,A -85,B 0,C 180,E1 13454.863,E2 13454.863} C_VEL
LIN {X 0,Y 306.393,Z 367.361,A -85,B 0,C 180,E1 13451.959,E2 13451.959} C_VEL
LIN {X 0,Y 294.454,Z 345.957,A -85,B 0,C 180,E1 13448.95,E2 13448.95} C_VEL
LIN {X 0,Y 289.228,Z 336.759,A -85,B 0,C 180,E1 13447.478,E2 13447.478} C_VEL
LIN {X 0,Y 283.078,Z 321.912,A -85,B 0,C 180,E1 13443.438,E2 13443.438} C_VEL
LIN {X 0,Y 281.913,Z 319.289,A -85,B 0,C 180,E1 13442.624,E2 13442.624} C_VEL
LIN {X 0,Y 282.497,Z 319.09,A -85,B 0,C 180,E1 13442.229,E2 13442.229} C_VEL
LIN {X 0,Y 283.327,Z 319.53,A -85,B 0,C 180,E1 13441.964,E2 13441.964} C_VEL
LIN {X 0,Y 288.214,Z 329.516,A -85,B 0,C 180,E1 13439.452,E2 13439.452} C_VEL
LIN {X 0,Y 294.105,Z 342.745,A -85,B 0,C 180,E1 13436.448,E2 13436.448} C_VEL
LIN {X 0,Y 300.291,Z 358.685,A -85,B 0,C 180,E1 13433.221,E2 13433.221} C_VEL
LIN {X 0,Y 305.477,Z 374.744,A -85,B 0,C 180,E1 13430.303,E2 13430.303} C_VEL
LIN {X 0,Y 305.898,Z 376.841,A -85,B 0,C 180,E1 13429.974,E2 13429.974} C_VEL
LIN {X 0,Y 301.217,Z 418.061,A -85,B 0,C 180,E1 13425.5,E2 13425.5} C_VEL
LIN {X 0,Y 296.144,Z 463.899,A -85,B 0,C 180,E1 13420.507,E2 13420.507} C_VEL
LIN {X 0,Y 294.131,Z 483.973,A -85,B 0,C 180,E1 13418.333,E2 13418.333} C_VEL
LIN {X 0,Y 296.153,Z 508.292,A -85,B 0,C 180,E1 13417.4,E2 13417.4} C_VEL
LIN {X 0,Y 291.612,Z 628.311,A -85,B 0,C 180,E1 13414.42,E2 13414.42} C_VEL
LIN {X 0,Y 290.461,Z 644.577,A -85,B 0,C 180,E1 13413.653,E2 13413.653} C_VEL
LIN {X 0,Y 288.844,Z 659.963,A -85,B 0,C 180,E1 13412.581,E2 13412.581} C_VEL
LIN {X 0,Y 286.828,Z 674.479,A -85,B 0,C 180,E1 13411.201,E2 13411.201} C_VEL
LIN {X 0,Y 284.4,Z 688.956,A -85,B 0,C 180,E1 13409.398,E2 13409.398} C_VEL
LIN {X 0,Y 281.941,Z 701.682,A -85,B 0,C 180,E1 13407.36,E2 13407.36} C_VEL
LIN {X 0,Y 279.398,Z 713.914,A -85,B 0,C 180,E1 13404.869,E2 13404.869} C_VEL
LIN {X 0,Y 277.25,Z 723.696,A -85,B 0,C 180,E1 13402.334,E2 13402.334} C_VEL
LIN {X 0,Y 275.277,Z 732.784,A -85,B 0,C 180,E1 13399.327,E2 13399.327} C_VEL
LIN {X 0,Y 273.835,Z 739.852,A -85,B 0,C 180,E1 13396.232,E2 13396.232} C_VEL
LIN {X 0,Y 272.879,Z 745.29,A -85,B 0,C 180,E1 13392.957,E2 13392.957} C_VEL
LIN {X 0,Y 272.485,Z 748.065,A -85,B 0,C 180,E1 13390.564,E2 13390.564} C_VEL
LIN {X 0,Y 271.339,Z 749.481,A -85,B 0,C 180,E1 13388.975,E2 13388.975} C_VEL
LIN {X 0,Y 267.308,Z 751.012,A -85,B 0,C 180,E1 13386.391,E2 13386.391} C_VEL
LIN {X 0,Y 264.503,Z 751.52,A -85,B 0,C 180,E1 13384.049,E2 13384.049} C_VEL
LIN {X 0,Y 264.253,Z 751.461,A -85,B 0,C 180,E1 13383.201,E2 13383.201} C_VEL
LIN {X 0,Y 264.517,Z 750.226,A -85,B 0,C 180,E1 13379.822,E2 13379.822} C_VEL
LIN {X 0,Y 265.178,Z 747.189,A -85,B 0,C 180,E1 13376.343,E2 13376.343} C_VEL
LIN {X 0,Y 266.324,Z 742.674,A -85,B 0,C 180,E1 13373.084,E2 13373.084} C_VEL
LIN {X 0,Y 268.09,Z 736.211,A -85,B 0,C 180,E1 13369.822,E2 13369.822} C_VEL
LIN {X 0,Y 270.38,Z 728.136,A -85,B 0,C 180,E1 13366.762,E2 13366.762} C_VEL
LIN {X 0,Y 273.042,Z 718.578,A -85,B 0,C 180,E1 13363.985,E2 13363.985} C_VEL
LIN {X 0,Y 276.104,Z 707.026,A -85,B 0,C 180,E1 13361.357,E2 13361.357} C_VEL
LIN {X 0,Y 278.939,Z 695.288,A -85,B 0,C 180,E1 13359.267,E2 13359.267} C_VEL
LIN {X 0,Y 281.852,Z 681.584,A -85,B 0,C 180,E1 13357.346,E2 13357.346} C_VEL
LIN {X 0,Y 284.332,Z 667.76,A -85,B 0,C 180,E1 13355.853,E2 13355.853} C_VEL
LIN {X 0,Y 286.547,Z 651.795,A -85,B 0,C 180,E1 13354.57,E2 13354.57} C_VEL
LIN {X 0,Y 288.086,Z 635.94,A -85,B 0,C 180,E1 13353.685,E2 13353.685} C_VEL
LIN {X 0,Y 289.074,Z 617.517,A -85,B 0,C 180,E1 13353.073,E2 13353.073} C_VEL
LIN {X 0,Y 293.842,Z 507.242,A -85,B 0,C 180,E1 13350.289,E2 13350.289} C_VEL
LIN {X 0,Y 291.897,Z 484.925,A -85,B 0,C 180,E1 13349.207,E2 13349.207} C_VEL
LIN {X 0,Y 297.347,Z 440.426,A -85,B 0,C 180,E1 13344.326,E2 13344.326} C_VEL
LIN {X 0,Y 302.688,Z 399.075,A -85,B 0,C 180,E1 13339.829,E2 13339.829} C_VEL
LIN {X 0,Y 304.731,Z 382.077,A -85,B 0,C 180,E1 13337.965,E2 13337.965} C_VEL
LIN {X 0,Y 300.846,Z 368.621,A -85,B 0,C 180,E1 13335.223,E2 13335.223} C_VEL
LIN {X 0,Y 296.367,Z 356.318,A -85,B 0,C 180,E1 13332.272,E2 13332.272} C_VEL
LIN {X 0,Y 292.051,Z 346.383,A -85,B 0,C 180,E1 13329.459,E2 13329.459} C_VEL
LIN {X 0,Y 288.167,Z 338.303,A -85,B 0,C 180,E1 13326.776,E2 13326.776} C_VEL
LIN {X 0,Y 285.708,Z 333.699,A -85,B 0,C 180,E1 13325.02,E2 13325.02} C_VEL
LIN {X 0,Y 284.125,Z 330.703,A -85,B 0,C 180,E1 13323.835,E2 13323.835} C_VEL
LIN {X 0,Y 281.48,Z 325.966,A -85,B 0,C 180,E1 13321.629,E2 13321.629} C_VEL
LIN {X 0,Y 279.059,Z 321.939,A -85,B 0,C 180,E1 13319.59,E2 13319.59} C_VEL
LIN {X 0,Y 278.421,Z 320.879,A -85,B 0,C 180,E1 13318.972,E2 13318.972} C_VEL
LIN {X 0,Y 276.082,Z 317.675,A -85,B 0,C 180,E1 13316.679,E2 13316.679} C_VEL
LIN {X 0,Y 275.114,Z 315.512,A -85,B 0,C 180,E1 13315.415,E2 13315.415} C_VEL
LIN {X 0,Y 272.087,Z 312.03,A -85,B 0,C 180,E1 13311.548,E2 13311.548} C_VEL
LIN {X 0,Y 271.128,Z 309.776,A -85,B 0,C 180,E1 13309.375,E2 13309.375} C_VEL
LIN {X 0,Y 269.324,Z 308.419,A -85,B 0,C 180,E1 13303.612,E2 13303.612} C_VEL
LIN {X 0,Y 270.346,Z 309.154,A -85,B 0,C 180,E1 13297.602,E2 13297.602} C_VEL
LIN {X 0,Y 270.762,Z 309.633,A -85,B 0,C 180,E1 13296.612,E2 13296.612} C_VEL
LIN {X 0,Y 271.139,Z 313.626,A -85,B 0,C 180,E1 13294.675,E2 13294.675} C_VEL
LIN {X 0,Y 275.742,Z 323.281,A -85,B 0,C 180,E1 13291.699,E2 13291.699} C_VEL
LIN {X 0,Y 287.772,Z 342.313,A -85,B 0,C 180,E1 13288.21,E2 13288.21} C_VEL
LIN {X 0,Y 301.06,Z 364.388,A -85,B 0,C 180,E1 13284.758,E2 13284.758} C_VEL
LIN {X 0,Y 315.589,Z 390.323,A -85,B 0,C 180,E1 13281.323,E2 13281.323} C_VEL
LIN {X 0,Y 317.619,Z 394.628,A -85,B 0,C 180,E1 13280.845,E2 13280.845} C_VEL
LIN {X 0,Y 302.389,Z 575.956,A -85,B 0,C 180,E1 13275.338,E2 13275.338} C_VEL
LIN {X 0,Y 299.775,Z 597.094,A -85,B 0,C 180,E1 13274.383,E2 13274.383} C_VEL
LIN {X 0,Y 296.47,Z 618.357,A -85,B 0,C 180,E1 13273.07,E2 13273.07} C_VEL
LIN {X 0,Y 292.818,Z 638.227,A -85,B 0,C 180,E1 13271.482,E2 13271.482} C_VEL
LIN {X 0,Y 288.629,Z 658.3,A -85,B 0,C 180,E1 13269.454,E2 13269.454} C_VEL
LIN {X 0,Y 284.486,Z 676.419,A -85,B 0,C 180,E1 13267.191,E2 13267.191} C_VEL
LIN {X 0,Y 280.294,Z 693.704,A -85,B 0,C 180,E1 13264.551,E2 13264.551} C_VEL
LIN {X 0,Y 276.223,Z 709.913,A -85,B 0,C 180,E1 13261.534,E2 13261.534} C_VEL
LIN {X 0,Y 272.596,Z 724.476,A -85,B 0,C 180,E1 13258.237,E2 13258.237} C_VEL
LIN {X 0,Y 269.51,Z 737.495,A -85,B 0,C 180,E1 13254.644,E2 13254.644} C_VEL
LIN {X 0,Y 267.122,Z 748.76,A -85,B 0,C 180,E1 13250.827,E2 13250.827} C_VEL
LIN {X 0,Y 265.488,Z 758.169,A -85,B 0,C 180,E1 13246.855,E2 13246.855} C_VEL
LIN {X 0,Y 264.401,Z 767.852,A -85,B 0,C 180,E1 13241.644,E2 13241.644} C_VEL
LIN {X 0,Y 264.19,Z 772.658,A -85,B 0,C 180,E1 13238.266,E2 13238.266} C_VEL
LIN {X 0,Y 264.168,Z 775.682,A -85,B 0,C 180,E1 13234.992,E2 13234.992} C_VEL
LIN {X 0,Y 264.23,Z 777.064,A -85,B 0,C 180,E1 13231.732,E2 13231.732} C_VEL
LIN {X 0,Y 264.177,Z 777.43,A -85,B 0,C 180,E1 13227.395,E2 13227.395} C_VEL
LIN {X 0,Y 264.077,Z 776.453,A -85,B 0,C 180,E1 13223.476,E2 13223.476} C_VEL
LIN {X 0,Y 264.221,Z 773.841,A -85,B 0,C 180,E1 13219.312,E2 13219.312} C_VEL
LIN {X 0,Y 265.035,Z 769.328,A -85,B 0,C 180,E1 13214.91,E2 13214.91} C_VEL
LIN {X 0,Y 266.946,Z 762.598,A -85,B 0,C 180,E1 13210.298,E2 13210.298} C_VEL
LIN {X 0,Y 270.168,Z 753.796,A -85,B 0,C 180,E1 13205.743,E2 13205.743} C_VEL
LIN {X 0,Y 274.854,Z 742.845,A -85,B 0,C 180,E1 13201.3,E2 13201.3} C_VEL
LIN {X 0,Y 280.928,Z 729.973,A -85,B 0,C 180,E1 13197.134,E2 13197.134} C_VEL
LIN {X 0,Y 288.198,Z 715.598,A -85,B 0,C 180,E1 13193.362,E2 13193.362} C_VEL
LIN {X 0,Y 297.183,Z 698.695,A -85,B 0,C 180,E1 13189.759,E2 13189.759} C_VEL
LIN {X 0,Y 307.868,Z 679.659,A -85,B 0,C 180,E1 13186.486,E2 13186.486} C_VEL
LIN {X 0,Y 319.374,Z 660.145,A -85,B 0,C 180,E1 13183.809,E2 13183.809} C_VEL
LIN {X 0,Y 325.765,Z 649.611,A -85,B 0,C 180,E1 13182.586,E2 13182.586} C_VEL
LIN {X 0,Y 314.262,Z 666.991,A -85,B 0,C 180,E1 13180.23,E2 13180.23} C_VEL
LIN {X 0,Y 303.398,Z 683.845,A -85,B 0,C 180,E1 13177.327,E2 13177.327} C_VEL
LIN {X 0,Y 293.68,Z 699.52,A -85,B 0,C 180,E1 13173.941,E2 13173.941} C_VEL
LIN {X 0,Y 285.522,Z 712.972,A -85,B 0,C 180,E1 13170.282,E2 13170.282} C_VEL
LIN {X 0,Y 278.856,Z 724.281,A -85,B 0,C 180,E1 13166.398,E2 13166.398} C_VEL
LIN {X 0,Y 273.596,Z 733.507,A -85,B 0,C 180,E1 13162.337,E2 13162.337} C_VEL
LIN {X 0,Y 269.833,Z 740.386,A -85,B 0,C 180,E1 13158.358,E2 13158.358} C_VEL
LIN {X 0,Y 267.139,Z 745.587,A -85,B 0,C 180,E1 13154.205,E2 13154.205} C_VEL
LIN {X 0,Y 265.515,Z 748.851,A -85,B 0,C 180,E1 13150.194,E2 13150.194} C_VEL
LIN {X 0,Y 264.629,Z 750.502,A -85,B 0,C 180,E1 13146.072,E2 13146.072} C_VEL
LIN {X 0,Y 264.272,Z 750.466,A -85,B 0,C 180,E1 13142.167,E2 13142.167} C_VEL
LIN {X 0,Y 264.172,Z 748.978,A -85,B 0,C 180,E1 13138.481,E2 13138.481} C_VEL
LIN {X 0,Y 264.223,Z 746.024,A -85,B 0,C 180,E1 13134.788,E2 13134.788} C_VEL
LIN {X 0,Y 264.563,Z 741.161,A -85,B 0,C 180,E1 13130.866,E2 13130.866} C_VEL
LIN {X 0,Y 265.386,Z 734.396,A -85,B 0,C 180,E1 13126.934,E2 13126.934} C_VEL
LIN {X 0,Y 266.762,Z 726.114,A -85,B 0,C 180,E1 13123.225,E2 13123.225} C_VEL
LIN {X 0,Y 268.769,Z 716.047,A -85,B 0,C 180,E1 13119.637,E2 13119.637} C_VEL
LIN {X 0,Y 271.308,Z 704.577,A -85,B 0,C 180,E1 13116.315,E2 13116.315} C_VEL
LIN {X 0,Y 274.417,Z 691.206,A -85,B 0,C 180,E1 13113.14,E2 13113.14} C_VEL
LIN {X 0,Y 277.91,Z 676.283,A -85,B 0,C 180,E1 13110.231,E2 13110.231} C_VEL
LIN {X 0,Y 281.671,Z 659.728,A -85,B 0,C 180,E1 13107.586,E2 13107.586} C_VEL
LIN {X 0,Y 285.44,Z 642.18,A -85,B 0,C 180,E1 13105.303,E2 13105.303} C_VEL
LIN {X 0,Y 289.012,Z 623.955,A -85,B 0,C 180,E1 13103.384,E2 13103.384} C_VEL
LIN {X 0,Y 292.376,Z 604.552,A -85,B 0,C 180,E1 13101.757,E2 13101.757} C_VEL
LIN {X 0,Y 295.434,Z 583.617,A -85,B 0,C 180,E1 13100.414,E2 13100.414} C_VEL
LIN {X 0,Y 297.858,Z 562.33,A -85,B 0,C 180,E1 13099.438,E2 13099.438} C_VEL
LIN {X 0,Y 312.395,Z 394.234,A -85,B 0,C 180,E1 13094.056,E2 13094.056} C_VEL
LIN {X 0,Y 298.925,Z 368.327,A -85,B 0,C 180,E1 13090.808,E2 13090.808} C_VEL
LIN {X 0,Y 286.528,Z 346.299,A -85,B 0,C 180,E1 13087.546,E2 13087.546} C_VEL
LIN {X 0,Y 281.032,Z 336.77,A -85,B 0,C 180,E1 13085.949,E2 13085.949} C_VEL
LIN {X 0,Y 276.536,Z 325.965,A -85,B 0,C 180,E1 13082.846,E2 13082.846} C_VEL
LIN {X 0,Y 277.206,Z 325.934,A -85,B 0,C 180,E1 13082.431,E2 13082.431} C_VEL
LIN {X 0,Y 278.533,Z 326.078,A -85,B 0,C 180,E1 13082.092,E2 13082.092} C_VEL
LIN {X 0,Y 285.392,Z 340.857,A -85,B 0,C 180,E1 13078.432,E2 13078.432} C_VEL
LIN {X 0,Y 291.909,Z 357.019,A -85,B 0,C 180,E1 13074.919,E2 13074.919} C_VEL
LIN {X 0,Y 297.344,Z 372.904,A -85,B 0,C 180,E1 13071.859,E2 13071.859} C_VEL
LIN {X 0,Y 299.23,Z 379.812,A -85,B 0,C 180,E1 13070.654,E2 13070.654} C_VEL
LIN {X 0,Y 294.192,Z 422.409,A -85,B 0,C 180,E1 13065.981,E2 13065.981} C_VEL
LIN {X 0,Y 288.952,Z 467.762,A -85,B 0,C 180,E1 13060.973,E2 13060.973} C_VEL
LIN {X 0,Y 287.226,Z 484.319,A -85,B 0,C 180,E1 13059.153,E2 13059.153} C_VEL
LIN {X 0,Y 289.214,Z 509.1,A -85,B 0,C 180,E1 13058.173,E2 13058.173} C_VEL
LIN {X 0,Y 284.508,Z 628.629,A -85,B 0,C 180,E1 13055.149,E2 13055.149} C_VEL
LIN {X 0,Y 283.309,Z 644.913,A -85,B 0,C 180,E1 13054.366,E2 13054.366} C_VEL
LIN {X 0,Y 281.525,Z 661.149,A -85,B 0,C 180,E1 13053.204,E2 13053.204} C_VEL
LIN {X 0,Y 279.362,Z 675.851,A -85,B 0,C 180,E1 13051.746,E2 13051.746} C_VEL
LIN {X 0,Y 276.849,Z 690.156,A -85,B 0,C 180,E1 13049.899,E2 13049.899} C_VEL
LIN {X 0,Y 274.178,Z 703.264,A -85,B 0,C 180,E1 13047.703,E2 13047.703} C_VEL
LIN {X 0,Y 271.76,Z 714.369,A -85,B 0,C 180,E1 13045.36,E2 13045.36} C_VEL
LIN {X 0,Y 269.511,Z 724.138,A -85,B 0,C 180,E1 13042.756,E2 13042.756} C_VEL
LIN {X 0,Y 267.442,Z 733.22,A -85,B 0,C 180,E1 13039.665,E2 13039.665} C_VEL
LIN {X 0,Y 265.941,Z 740.196,A -85,B 0,C 180,E1 13036.523,E2 13036.523} C_VEL
LIN {X 0,Y 264.918,Z 745.708,A -85,B 0,C 180,E1 13033.108,E2 13033.108} C_VEL
LIN {X 0,Y 264.403,Z 749.31,A -85,B 0,C 180,E1 13029.693,E2 13029.693} C_VEL
LIN {X 0,Y 264.224,Z 751.237,A -85,B 0,C 180,E1 13026.118,E2 13026.118} C_VEL
LIN {X 0,Y 264.253,Z 751.461,A -85,B 0,C 180,E1 13023.201,E2 13023.201} C_VEL
LIN {X 0,Y 263.343,Z 751.16,A -85,B 0,C 180,E1 13021.529,E2 13021.529} C_VEL
LIN {X 0,Y 259.575,Z 749.852,A -85,B 0,C 180,E1 13018.715,E2 13018.715} C_VEL
LIN {X 0,Y 257.435,Z 748.046,A -85,B 0,C 180,E1 13016.438,E2 13016.438} C_VEL
LIN {X 0,Y 257.406,Z 747.146,A -85,B 0,C 180,E1 13015.589,E2 13015.589} C_VEL
LIN {X 0,Y 258.784,Z 742.152,A -85,B 0,C 180,E1 13012.101,E2 13012.101} C_VEL
LIN {X 0,Y 260.819,Z 735.313,A -85,B 0,C 180,E1 13008.711,E2 13008.711} C_VEL
LIN {X 0,Y 263.284,Z 727.137,A -85,B 0,C 180,E1 13005.676,E2 13005.676} C_VEL
LIN {X 0,Y 266.204,Z 717.225,A -85,B 0,C 180,E1 13002.832,E2 13002.832} C_VEL
LIN {X 0,Y 269.174,Z 706.501,A -85,B 0,C 180,E1 13000.41,E2 13000.41} C_VEL
LIN {X 0,Y 272.289,Z 694.083,A -85,B 0,C 180,E1 12998.208,E2 12998.208} C_VEL
LIN {X 0,Y 275.306,Z 680.345,A -85,B 0,C 180,E1 12996.299,E2 12996.299} C_VEL
LIN {X 0,Y 278.057,Z 665.112,A -85,B 0,C 180,E1 12994.701,E2 12994.701} C_VEL
LIN {X 0,Y 280.097,Z 650.585,A -85,B 0,C 180,E1 12993.561,E2 12993.561} C_VEL
LIN {X 0,Y 281.68,Z 634.016,A -85,B 0,C 180,E1 12992.672,E2 12992.672} C_VEL
LIN {X 0,Y 282.694,Z 614.707,A -85,B 0,C 180,E1 12992.065,E2 12992.065} C_VEL
LIN {X 0,Y 287.556,Z 508.326,A -85,B 0,C 180,E1 12989.331,E2 12989.331} C_VEL
LIN {X 0,Y 285.615,Z 485.555,A -85,B 0,C 180,E1 12988.204,E2 12988.204} C_VEL
LIN {X 0,Y 291.235,Z 441.939,A -85,B 0,C 180,E1 12983.362,E2 12983.362} C_VEL
LIN {X 0,Y 296.94,Z 400.103,A -85,B 0,C 180,E1 12978.759,E2 12978.759} C_VEL
LIN {X 0,Y 298.792,Z 385.556,A -85,B 0,C 180,E1 12977.127,E2 12977.127} C_VEL
LIN {X 0,Y 295.026,Z 372.369,A -85,B 0,C 180,E1 12974.325,E2 12974.325} C_VEL
LIN {X 0,Y 290.73,Z 360.298,A -85,B 0,C 180,E1 12971.306,E2 12971.306} C_VEL
LIN {X 0,Y 286.134,Z 349.446,A -85,B 0,C 180,E1 12968.036,E2 12968.036} C_VEL
LIN {X 0,Y 282.035,Z 341.18,A -85,B 0,C 180,E1 12965.038,E2 12965.038} C_VEL
LIN {X 0,Y 279.846,Z 337.032,A -85,B 0,C 180,E1 12963.278,E2 12963.278} C_VEL
LIN {X 0,Y 277.551,Z 332.713,A -85,B 0,C 180,E1 12961.239,E2 12961.239} C_VEL
LIN {X 0,Y 275.306,Z 328.719,A -85,B 0,C 180,E1 12959.168,E2 12959.168} C_VEL
LIN {X 0,Y 272.385,Z 324.11,A -85,B 0,C 180,E1 12956.001,E2 12956.001} C_VEL
LIN {X 0,Y 271.755,Z 322.71,A -85,B 0,C 180,E1 12955.146,E2 12955.146} C_VEL
LIN {X 0,Y 268.885,Z 319.004,A -85,B 0,C 180,E1 12951.016,E2 12951.016} C_VEL
LIN {X 0,Y 268.106,Z 317.079,A -85,B 0,C 180,E1 12949.036,E2 12949.036} C_VEL
LIN {X 0,Y 266.633,Z 315.935,A -85,B 0,C 180,E1 12942.976,E2 12942.976} C_VEL
LIN {X 0,Y 267.959,Z 316.873,A -85,B 0,C 180,E1 12937.109,E2 12937.109} C_VEL
LIN {X 0,Y 268.11,Z 322.342,A -85,B 0,C 180,E1 12934.368,E2 12934.368} C_VEL
LIN {X 0,Y 268.563,Z 325.134,A -85,B 0,C 180,E1 12933.166,E2 12933.166} C_VEL
LIN {X 0,Y 280.399,Z 343.647,A -85,B 0,C 180,E1 12929.58,E2 12929.58} C_VEL
LIN {X 0,Y 293.861,Z 366.106,A -85,B 0,C 180,E1 12925.906,E2 12925.906} C_VEL
LIN {X 0,Y 307.067,Z 389.595,A -85,B 0,C 180,E1 12922.637,E2 12922.637} C_VEL
LIN {X 0,Y 311.122,Z 397.45,A -85,B 0,C 180,E1 12921.676,E2 12921.676} C_VEL
LIN {X 0,Y 295.469,Z 576.065,A -85,B 0,C 180,E1 12916.108,E2 12916.108} C_VEL
LIN {X 0,Y 292.753,Z 597.216,A -85,B 0,C 180,E1 12915.124,E2 12915.124} C_VEL
LIN {X 0,Y 289.439,Z 617.893,A -85,B 0,C 180,E1 12913.82,E2 12913.82} C_VEL
LIN {X 0,Y 285.489,Z 638.664,A -85,B 0,C 180,E1 12912.116,E2 12912.116} C_VEL
LIN {X 0,Y 281.43,Z 657.558,A -85,B 0,C 180,E1 12910.168,E2 12910.168} C_VEL
LIN {X 0,Y 277.005,Z 676.334,A -85,B 0,C 180,E1 12907.77,E2 12907.77} C_VEL
LIN {X 0,Y 272.656,Z 693.714,A -85,B 0,C 180,E1 12905.043,E2 12905.043} C_VEL
LIN {X 0,Y 268.576,Z 709.476,A -85,B 0,C 180,E1 12902.036,E2 12902.036} C_VEL
LIN {X 0,Y 264.829,Z 724.067,A -85,B 0,C 180,E1 12898.649,E2 12898.649} C_VEL
LIN {X 0,Y 261.74,Z 736.697,A -85,B 0,C 180,E1 12895.086,E2 12895.086} C_VEL
LIN {X 0,Y 259.298,Z 747.805,A -85,B 0,C 180,E1 12891.249,E2 12891.249} C_VEL
LIN {X 0,Y 257.574,Z 757.323,A -85,B 0,C 180,E1 12887.156,E2 12887.156} C_VEL
LIN {X 0,Y 256.562,Z 766.176,A -85,B 0,C 180,E1 12882.832,E2 12882.832} C_VEL
LIN {X 0,Y 256.224,Z 771.289,A -85,B 0,C 180,E1 12879.43,E2 12879.43} C_VEL
LIN {X 0,Y 256.172,Z 774.841,A -85,B 0,C 180,E1 12875.822,E2 12875.822} C_VEL
LIN {X 0,Y 256.225,Z 776.542,A -85,B 0,C 180,E1 12872.458,E2 12872.458} C_VEL
LIN {X 0,Y 256.224,Z 776.895,A -85,B 0,C 180,E1 12868.209,E2 12868.209} C_VEL
LIN {X 0,Y 256.095,Z 776.47,A -85,B 0,C 180,E1 12864.396,E2 12864.396} C_VEL
LIN {X 0,Y 256.135,Z 774.535,A -85,B 0,C 180,E1 12860.334,E2 12860.334} C_VEL
LIN {X 0,Y 256.782,Z 770.746,A -85,B 0,C 180,E1 12855.823,E2 12855.823} C_VEL
LIN {X 0,Y 258.426,Z 765.131,A -85,B 0,C 180,E1 12851.266,E2 12851.266} C_VEL
LIN {X 0,Y 261.437,Z 757.306,A -85,B 0,C 180,E1 12846.56,E2 12846.56} C_VEL
LIN {X 0,Y 265.948,Z 747.434,A -85,B 0,C 180,E1 12841.967,E2 12841.967} C_VEL
LIN {X 0,Y 272.081,Z 735.449,A -85,B 0,C 180,E1 12837.55,E2 12837.55} C_VEL
LIN {X 0,Y 279.493,Z 722.038,A -85,B 0,C 180,E1 12833.567,E2 12833.567} C_VEL
LIN {X 0,Y 288.993,Z 705.853,A -85,B 0,C 180,E1 12829.683,E2 12829.683} C_VEL
LIN {X 0,Y 299.761,Z 688.525,A -85,B 0,C 180,E1 12826.332,E2 12826.332} C_VEL
LIN {X 0,Y 311.664,Z 670.423,A -85,B 0,C 180,E1 12823.526,E2 12823.526} C_VEL
LIN {X 0,Y 316.699,Z 662.999,A -85,B 0,C 180,E1 12822.533,E2 12822.533} C_VEL
LIN {X 0,Y 304.303,Z 679.759,A -85,B 0,C 180,E1 12819.845,E2 12819.845} C_VEL
LIN {X 0,Y 293.114,Z 695.355,A -85,B 0,C 180,E1 12816.651,E2 12816.651} C_VEL
LIN {X 0,Y 283.18,Z 709.698,A -85,B 0,C 180,E1 12812.938,E2 12812.938} C_VEL
LIN {X 0,Y 275.344,Z 721.405,A -85,B 0,C 180,E1 12809.116,E2 12809.116} C_VEL
LIN {X 0,Y 269.011,Z 731.149,A -85,B 0,C 180,E1 12805.069,E2 12805.069} C_VEL
LIN {X 0,Y 264.108,Z 738.947,A -85,B 0,C 180,E1 12800.846,E2 12800.846} C_VEL
LIN {X 0,Y 260.554,Z 744.818,A -85,B 0,C 180,E1 12796.497,E2 12796.497} C_VEL
LIN {X 0,Y 258.222,Z 748.792,A -85,B 0,C 180,E1 12792.068,E2 12792.068} C_VEL
LIN {X 0,Y 256.91,Z 750.895,A -85,B 0,C 180,E1 12787.603,E2 12787.603} C_VEL
LIN {X 0,Y 256.377,Z 751.195,A -85,B 0,C 180,E1 12783.577,E2 12783.577} C_VEL
LIN {X 0,Y 256.196,Z 749.887,A -85,B 0,C 180,E1 12779.552,E2 12779.552} C_VEL
LIN {X 0,Y 256.191,Z 747.15,A -85,B 0,C 180,E1 12775.747,E2 12775.747} C_VEL
LIN {X 0,Y 256.434,Z 742.885,A -85,B 0,C 180,E1 12771.93,E2 12771.93} C_VEL
LIN {X 0,Y 257.125,Z 736.57,A -85,B 0,C 180,E1 12767.878,E2 12767.878} C_VEL
LIN {X 0,Y 258.365,Z 728.743,A -85,B 0,C 180,E1 12764.051,E2 12764.051} C_VEL
LIN {X 0,Y 260.321,Z 718.846,A -85,B 0,C 180,E1 12760.227,E2 12760.227} C_VEL
LIN {X 0,Y 262.858,Z 707.504,A -85,B 0,C 180,E1 12756.696,E2 12756.696} C_VEL
LIN {X 0,Y 265.921,Z 694.644,A -85,B 0,C 180,E1 12753.42,E2 12753.42} C_VEL
LIN {X 0,Y 269.39,Z 680.327,A -85,B 0,C 180,E1 12750.419,E2 12750.419} C_VEL
LIN {X 0,Y 273.303,Z 663.874,A -85,B 0,C 180,E1 12747.59,E2 12747.59} C_VEL
LIN {X 0,Y 277.26,Z 646.249,A -85,B 0,C 180,E1 12745.138,E2 12745.138} C_VEL
LIN {X 0,Y 281.09,Z 627.597,A -85,B 0,C 180,E1 12743.047,E2 12743.047} C_VEL
LIN {X 0,Y 284.671,Z 608.006,A -85,B 0,C 180,E1 12741.302,E2 12741.302} C_VEL
LIN {X 0,Y 287.862,Z 587.393,A -85,B 0,C 180,E1 12739.885,E2 12739.885} C_VEL
LIN {X 0,Y 290.507,Z 566.391,A -85,B 0,C 180,E1 12738.825,E2 12738.825} C_VEL
LIN {X 0,Y 299.392,Z 466.167,A -85,B 0,C 180,E1 12735.431,E2 12735.431} C_VEL
LIN {X 0,Y 305.766,Z 396.925,A -85,B 0,C 180,E1 12733.211,E2 12733.211} C_VEL
LIN {X 0,Y 293.128,Z 372.457,A -85,B 0,C 180,E1 12730.048,E2 12730.048} C_VEL
LIN {X 0,Y 281.063,Z 350.849,A -85,B 0,C 180,E1 12726.767,E2 12726.767} C_VEL
LIN {X 0,Y 272.665,Z 336.54,A -85,B 0,C 180,E1 12724.258,E2 12724.258} C_VEL
LIN {X 0,Y 271.176,Z 332.651,A -85,B 0,C 180,E1 12723.035,E2 12723.035} C_VEL
LIN {X 0,Y 272.605,Z 332.766,A -85,B 0,C 180,E1 12722.477,E2 12722.477} C_VEL
LIN {X 0,Y 273.848,Z 333.25,A -85,B 0,C 180,E1 12722.104,E2 12722.104} C_VEL
LIN {X 0,Y 279.927,Z 346.608,A -85,B 0,C 180,E1 12718.75,E2 12718.75} C_VEL
LIN {X 0,Y 286.015,Z 361.966,A -85,B 0,C 180,E1 12715.358,E2 12715.358} C_VEL
LIN {X 0,Y 291.59,Z 378.781,A -85,B 0,C 180,E1 12712.066,E2 12712.066} C_VEL
LIN {X 0,Y 292.582,Z 382.952,A -85,B 0,C 180,E1 12711.345,E2 12711.345} C_VEL
LIN {X 0,Y 287.272,Z 425.798,A -85,B 0,C 180,E1 12706.585,E2 12706.585} C_VEL
LIN {X 0,Y 281.887,Z 470.765,A -85,B 0,C 180,E1 12701.563,E2 12701.563} C_VEL
LIN {X 0,Y 280.377,Z 484.638,A -85,B 0,C 180,E1 12700.014,E2 12700.014} C_VEL
LIN {X 0,Y 282.329,Z 509.85,A -85,B 0,C 180,E1 12698.983,E2 12698.983} C_VEL
LIN {X 0,Y 277.427,Z 629.056,A -85,B 0,C 180,E1 12695.904,E2 12695.904} C_VEL
LIN {X 0,Y 276.177,Z 645.328,A -85,B 0,C 180,E1 12695.104,E2 12695.104} C_VEL
LIN {X 0,Y 274.405,Z 660.879,A -85,B 0,C 180,E1 12693.972,E2 12693.972} C_VEL
LIN {X 0,Y 272.222,Z 675.36,A -85,B 0,C 180,E1 12692.528,E2 12692.528} C_VEL
LIN {X 0,Y 269.588,Z 689.834,A -85,B 0,C 180,E1 12690.64,E2 12690.64} C_VEL
LIN {X 0,Y 266.915,Z 702.546,A -85,B 0,C 180,E1 12688.5,E2 12688.5} C_VEL
LIN {X 0,Y 264.139,Z 714.779,A -85,B 0,C 180,E1 12685.878,E2 12685.878} C_VEL
LIN {X 0,Y 261.785,Z 724.548,A -85,B 0,C 180,E1 12683.203,E2 12683.203} C_VEL
LIN {X 0,Y 259.615,Z 733.633,A -85,B 0,C 180,E1 12680.022,E2 12680.022} C_VEL
LIN {X 0,Y 258.037,Z 740.606,A -85,B 0,C 180,E1 12676.787,E2 12676.787} C_VEL
LIN {X 0,Y 256.943,Z 746.215,A -85,B 0,C 180,E1 12673.194,E2 12673.194} C_VEL
LIN {X 0,Y 256.412,Z 749.748,A -85,B 0,C 180,E1 12669.696,E2 12669.696} C_VEL
LIN {X 0,Y 256.231,Z 751.673,A -85,B 0,C 180,E1 12665.941,E2 12665.941} C_VEL
LIN {X 0,Y 256.302,Z 751.729,A -85,B 0,C 180,E1 12662.343,E2 12662.343} C_VEL
LIN {X 0,Y 256.718,Z 749.922,A -85,B 0,C 180,E1 12658.536,E2 12658.536} C_VEL
LIN {X 0,Y 257.406,Z 747.146,A -85,B 0,C 180,E1 12655.589,E2 12655.589} C_VEL
LIN {X 0,Y 256.996,Z 745.207,A -85,B 0,C 180,E1 12653.917,E2 12653.917} C_VEL
LIN {X 0,Y 253.978,Z 740.913,A -85,B 0,C 180,E1 12650.871,E2 12650.871} C_VEL
LIN {X 0,Y 252.927,Z 737.614,A -85,B 0,C 180,E1 12649.011,E2 12649.011} C_VEL
LIN {X 0,Y 253.22,Z 735.69,A -85,B 0,C 180,E1 12648.102,E2 12648.102} C_VEL
LIN {X 0,Y 255.85,Z 727.502,A -85,B 0,C 180,E1 12644.985,E2 12644.985} C_VEL
LIN {X 0,Y 258.986,Z 717.445,A -85,B 0,C 180,E1 12642.034,E2 12642.034} C_VEL
LIN {X 0,Y 262.25,Z 706.223,A -85,B 0,C 180,E1 12639.466,E2 12639.466} C_VEL
LIN {X 0,Y 265.744,Z 692.935,A -85,B 0,C 180,E1 12637.099,E2 12637.099} C_VEL
LIN {X 0,Y 268.866,Z 679.065,A -85,B 0,C 180,E1 12635.2,E2 12635.2} C_VEL
LIN {X 0,Y 271.687,Z 663.938,A -85,B 0,C 180,E1 12633.624,E2 12633.624} C_VEL
LIN {X 0,Y 273.868,Z 648.2,A -85,B 0,C 180,E1 12632.437,E2 12632.437} C_VEL
LIN {X 0,Y 275.42,Z 631.652,A -85,B 0,C 180,E1 12631.589,E2 12631.589} C_VEL
LIN {X 0,Y 278.117,Z 576.528,A -85,B 0,C 180,E1 12630.083,E2 12630.083} C_VEL
LIN {X 0,Y 281.382,Z 509.252,A -85,B 0,C 180,E1 12628.313,E2 12628.313} C_VEL
LIN {X 0,Y 279.555,Z 485.416,A -85,B 0,C 180,E1 12627.061,E2 12627.061} C_VEL
LIN {X 0,Y 285.902,Z 439.143,A -85,B 0,C 180,E1 12621.868,E2 12621.868} C_VEL
LIN {X 0,Y 292.228,Z 395.584,A -85,B 0,C 180,E1 12617.011,E2 12617.011} C_VEL
LIN {X 0,Y 293.049,Z 389.555,A -85,B 0,C 180,E1 12616.35,E2 12616.35} C_VEL
LIN {X 0,Y 289.558,Z 376.947,A -85,B 0,C 180,E1 12613.581,E2 12613.581} C_VEL
LIN {X 0,Y 285.465,Z 365.026,A -85,B 0,C 180,E1 12610.495,E2 12610.495} C_VEL
LIN {X 0,Y 281.342,Z 355.057,A -85,B 0,C 180,E1 12607.351,E2 12607.351} C_VEL
LIN {X 0,Y 277.52,Z 347.06,A -85,B 0,C 180,E1 12604.34,E2 12604.34} C_VEL
LIN {X 0,Y 275.656,Z 343.37,A -85,B 0,C 180,E1 12602.703,E2 12602.703} C_VEL
LIN {X 0,Y 273.619,Z 339.446,A -85,B 0,C 180,E1 12600.838,E2 12600.838} C_VEL
LIN {X 0,Y 271.208,Z 334.904,A -85,B 0,C 180,E1 12598.311,E2 12598.311} C_VEL
LIN {X 0,Y 269.01,Z 331.316,A -85,B 0,C 180,E1 12595.738,E2 12595.738} C_VEL
LIN {X 0,Y 268.402,Z 329.91,A -85,B 0,C 180,E1 12594.871,E2 12594.871} C_VEL
LIN {X 0,Y 265.797,Z 326.228,A -85,B 0,C 180,E1 12590.692,E2 12590.692} C_VEL
LIN {X 0,Y 265.181,Z 324.503,A -85,B 0,C 180,E1 12588.914,E2 12588.914} C_VEL
LIN {X 0,Y 263.927,Z 323.468,A -85,B 0,C 180,E1 12582.814,E2 12582.814} C_VEL
LIN {X 0,Y 265.171,Z 324.337,A -85,B 0,C 180,E1 12577.481,E2 12577.481} C_VEL
LIN {X 0,Y 265.167,Z 329.151,A -85,B 0,C 180,E1 12575.02,E2 12575.02} C_VEL
LIN {X 0,Y 265.422,Z 332.988,A -85,B 0,C 180,E1 12573.428,E2 12573.428} C_VEL
LIN {X 0,Y 277.388,Z 352.176,A -85,B 0,C 180,E1 12569.694,E2 12569.694} C_VEL
LIN {X 0,Y 291.163,Z 375.535,A -85,B 0,C 180,E1 12565.903,E2 12565.903} C_VEL
LIN {X 0,Y 304.653,Z 399.967,A -85,B 0,C 180,E1 12562.544,E2 12562.544} C_VEL
LIN {X 0,Y 288.575,Z 575.961,A -85,B 0,C 180,E1 12556.904,E2 12556.904} C_VEL
LIN {X 0,Y 285.646,Z 597.916,A -85,B 0,C 180,E1 12555.85,E2 12555.85} C_VEL
LIN {X 0,Y 282.271,Z 618.214,A -85,B 0,C 180,E1 12554.532,E2 12554.532} C_VEL
LIN {X 0,Y 278.195,Z 638.944,A -85,B 0,C 180,E1 12552.784,E2 12552.784} C_VEL
LIN {X 0,Y 274,Z 657.836,A -85,B 0,C 180,E1 12550.779,E2 12550.779} C_VEL
LIN {X 0,Y 269.634,Z 675.826,A -85,B 0,C 180,E1 12548.427,E2 12548.427} C_VEL
LIN {X 0,Y 265.139,Z 693.255,A -85,B 0,C 180,E1 12545.632,E2 12545.632} C_VEL
LIN {X 0,Y 260.913,Z 709.095,A -85,B 0,C 180,E1 12542.535,E2 12542.535} C_VEL
LIN {X 0,Y 257.077,Z 723.582,A -85,B 0,C 180,E1 12539.086,E2 12539.086} C_VEL
LIN {X 0,Y 253.884,Z 736.239,A -85,B 0,C 180,E1 12535.418,E2 12535.418} C_VEL
LIN {X 0,Y 251.35,Z 747.43,A -85,B 0,C 180,E1 12531.435,E2 12531.435} C_VEL
LIN {X 0,Y 249.316,Z 760.034,A -85,B 0,C 180,E1 12526.301,E2 12526.301} C_VEL
LIN {X 0,Y 248.554,Z 766.708,A -85,B 0,C 180,E1 12522.78,E2 12522.78} C_VEL
LIN {X 0,Y 248.207,Z 771.783,A -85,B 0,C 180,E1 12519.036,E2 12519.036} C_VEL
LIN {X 0,Y 248.173,Z 774.842,A -85,B 0,C 180,E1 12515.546,E2 12515.546} C_VEL
LIN {X 0,Y 248.24,Z 776.268,A -85,B 0,C 180,E1 12512.075,E2 12512.075} C_VEL
LIN {X 0,Y 248.223,Z 776.367,A -85,B 0,C 180,E1 12507.689,E2 12507.689} C_VEL
LIN {X 0,Y 248.094,Z 775.911,A -85,B 0,C 180,E1 12503.751,E2 12503.751} C_VEL
LIN {X 0,Y 248.218,Z 773.809,A -85,B 0,C 180,E1 12499.319,E2 12499.319} C_VEL
LIN {X 0,Y 249.171,Z 769.632,A -85,B 0,C 180,E1 12494.375,E2 12494.375} C_VEL
LIN {X 0,Y 251.338,Z 763.593,A -85,B 0,C 180,E1 12489.506,E2 12489.506} C_VEL
LIN {X 0,Y 254.987,Z 755.598,A -85,B 0,C 180,E1 12484.694,E2 12484.694} C_VEL
LIN {X 0,Y 260.25,Z 745.641,A -85,B 0,C 180,E1 12480.034,E2 12480.034} C_VEL
LIN {X 0,Y 267.22,Z 733.705,A -85,B 0,C 180,E1 12475.596,E2 12475.596} C_VEL
LIN {X 0,Y 275.965,Z 719.805,A -85,B 0,C 180,E1 12471.449,E2 12471.449} C_VEL
LIN {X 0,Y 287.073,Z 703.228,A -85,B 0,C 180,E1 12467.49,E2 12467.49} C_VEL
LIN {X 0,Y 299.64,Z 685.661,A -85,B 0,C 180,E1 12464.155,E2 12464.155} C_VEL
LIN {X 0,Y 307.526,Z 675.142,A -85,B 0,C 180,E1 12462.466,E2 12462.466} C_VEL
LIN {X 0,Y 294.888,Z 690.385,A -85,B 0,C 180,E1 12459.6,E2 12459.6} C_VEL
LIN {X 0,Y 282.713,Z 705.662,A -85,B 0,C 180,E1 12455.912,E2 12455.912} C_VEL
LIN {X 0,Y 272.716,Z 718.764,A -85,B 0,C 180,E1 12451.866,E2 12451.866} C_VEL
LIN {X 0,Y 264.863,Z 729.274,A -85,B 0,C 180,E1 12447.666,E2 12447.666} C_VEL
LIN {X 0,Y 258.947,Z 737.428,A -85,B 0,C 180,E1 12443.434,E2 12443.434} C_VEL
LIN {X 0,Y 254.487,Z 743.76,A -85,B 0,C 180,E1 12439.031,E2 12439.031} C_VEL
LIN {X 0,Y 251.395,Z 748.261,A -85,B 0,C 180,E1 12434.51,E2 12434.51} C_VEL
LIN {X 0,Y 249.503,Z 750.937,A -85,B 0,C 180,E1 12429.922,E2 12429.922} C_VEL
LIN {X 0,Y 248.594,Z 751.782,A -85,B 0,C 180,E1 12425.539,E2 12425.539} C_VEL
LIN {X 0,Y 248.261,Z 751.006,A -85,B 0,C 180,E1 12421.384,E2 12421.384} C_VEL
LIN {X 0,Y 248.173,Z 748.831,A -85,B 0,C 180,E1 12417.459,E2 12417.459} C_VEL
LIN {X 0,Y 248.31,Z 744.859,A -85,B 0,C 180,E1 12413.293,E2 12413.293} C_VEL
LIN {X 0,Y 248.853,Z 739.068,A -85,B 0,C 180,E1 12409.114,E2 12409.114} C_VEL
LIN {X 0,Y 250.004,Z 731.303,A -85,B 0,C 180,E1 12404.931,E2 12404.931} C_VEL
LIN {X 0,Y 251.806,Z 721.935,A -85,B 0,C 180,E1 12400.997,E2 12400.997} C_VEL
LIN {X 0,Y 254.234,Z 711.077,A -85,B 0,C 180,E1 12397.329,E2 12397.329} C_VEL
LIN {X 0,Y 257.275,Z 698.511,A -85,B 0,C 180,E1 12393.867,E2 12393.867} C_VEL
LIN {X 0,Y 260.864,Z 684.098,A -85,B 0,C 180,E1 12390.618,E2 12390.618} C_VEL
LIN {X 0,Y 264.765,Z 668.262,A -85,B 0,C 180,E1 12387.698,E2 12387.698} C_VEL
LIN {X 0,Y 268.892,Z 650.709,A -85,B 0,C 180,E1 12385.064,E2 12385.064} C_VEL
LIN {X 0,Y 272.949,Z 632.099,A -85,B 0,C 180,E1 12382.812,E2 12382.812} C_VEL
LIN {X 0,Y 276.751,Z 612.591,A -85,B 0,C 180,E1 12380.929,E2 12380.929} C_VEL
LIN {X 0,Y 280.116,Z 592.33,A -85,B 0,C 180,E1 12379.417,E2 12379.417} C_VEL
LIN {X 0,Y 283.01,Z 571.163,A -85,B 0,C 180,E1 12378.243,E2 12378.243} C_VEL
LIN {X 0,Y 285.913,Z 541.776,A -85,B 0,C 180,E1 12377.115,E2 12377.115} C_VEL
LIN {X 0,Y 299.252,Z 399.79,A -85,B 0,C 180,E1 12372.363,E2 12372.363} C_VEL
LIN {X 0,Y 287.388,Z 376.669,A -85,B 0,C 180,E1 12369.289,E2 12369.289} C_VEL
LIN {X 0,Y 275.771,Z 355.743,A -85,B 0,C 180,E1 12366.036,E2 12366.036} C_VEL
LIN {X 0,Y 266.659,Z 340.131,A -85,B 0,C 180,E1 12363.194,E2 12363.194} C_VEL
LIN {X 0,Y 266.891,Z 339.624,A -85,B 0,C 180,E1 12362.846,E2 12362.846} C_VEL
LIN {X 0,Y 268.978,Z 339.864,A -85,B 0,C 180,E1 12362.254,E2 12362.254} C_VEL
LIN {X 0,Y 275.266,Z 354.159,A -85,B 0,C 180,E1 12358.653,E2 12358.653} C_VEL
LIN {X 0,Y 281.019,Z 369.487,A -85,B 0,C 180,E1 12355.277,E2 12355.277} C_VEL
LIN {X 0,Y 285.974,Z 385.172,A -85,B 0,C 180,E1 12352.187,E2 12352.187} C_VEL
LIN {X 0,Y 281.647,Z 419.515,A -85,B 0,C 180,E1 12348.313,E2 12348.313} C_VEL
LIN {X 0,Y 275.942,Z 464.782,A -85,B 0,C 180,E1 12343.198,E2 12343.198} C_VEL
LIN {X 0,Y 273.579,Z 484.324,A -85,B 0,C 180,E1 12340.958,E2 12340.958} C_VEL
LIN {X 0,Y 275.499,Z 510.719,A -85,B 0,C 180,E1 12339.83,E2 12339.83} C_VEL
LIN {X 0,Y 270.405,Z 629.316,A -85,B 0,C 180,E1 12336.704,E2 12336.704} C_VEL
LIN {X 0,Y 269.114,Z 645.535,A -85,B 0,C 180,E1 12335.893,E2 12335.893} C_VEL
LIN {X 0,Y 267.249,Z 661.287,A -85,B 0,C 180,E1 12334.724,E2 12334.724} C_VEL
LIN {X 0,Y 264.975,Z 675.763,A -85,B 0,C 180,E1 12333.247,E2 12333.247} C_VEL
LIN {X 0,Y 262.231,Z 690.238,A -85,B 0,C 180,E1 12331.313,E2 12331.313} C_VEL
LIN {X 0,Y 259.442,Z 702.948,A -85,B 0,C 180,E1 12329.119,E2 12329.119} C_VEL
LIN {X 0,Y 256.54,Z 715.184,A -85,B 0,C 180,E1 12326.427,E2 12326.427} C_VEL
LIN {X 0,Y 253.89,Z 725.671,A -85,B 0,C 180,E1 12323.445,E2 12323.445} C_VEL
LIN {X 0,Y 251.798,Z 734.038,A -85,B 0,C 180,E1 12320.402,E2 12320.402} C_VEL
LIN {X 0,Y 250.137,Z 741.007,A -85,B 0,C 180,E1 12317.068,E2 12317.068} C_VEL
LIN {X 0,Y 249.001,Z 746.517,A -85,B 0,C 180,E1 12313.438,E2 12313.438} C_VEL
LIN {X 0,Y 248.451,Z 749.972,A -85,B 0,C 180,E1 12310,E2 12310} C_VEL
LIN {X 0,Y 248.243,Z 751.951,A -85,B 0,C 180,E1 12306.251,E2 12306.251} C_VEL
LIN {X 0,Y 248.296,Z 752.234,A -85,B 0,C 180,E1 12302.676,E2 12302.676} C_VEL
LIN {X 0,Y 248.669,Z 750.756,A -85,B 0,C 180,E1 12298.921,E2 12298.921} C_VEL
LIN {X 0,Y 249.585,Z 747.388,A -85,B 0,C 180,E1 12295.053,E2 12295.053} C_VEL
LIN {X 0,Y 251.035,Z 742.53,A -85,B 0,C 180,E1 12291.59,E2 12291.59} C_VEL
LIN {X 0,Y 253.22,Z 735.69,A -85,B 0,C 180,E1 12288.102,E2 12288.102} C_VEL
LIN {X 0,Y 253.462,Z 732.181,A -85,B 0,C 180,E1 12286.536,E2 12286.536} C_VEL
LIN {X 0,Y 251.407,Z 724.108,A -85,B 0,C 180,E1 12283.23,E2 12283.23} C_VEL
LIN {X 0,Y 251.346,Z 719.743,A -85,B 0,C 180,E1 12281.763,E2 12281.763} C_VEL
LIN {X 0,Y 251.845,Z 717.662,A -85,B 0,C 180,E1 12281.176,E2 12281.176} C_VEL
LIN {X 0,Y 255.273,Z 706.473,A -85,B 0,C 180,E1 12278.568,E2 12278.568} C_VEL
LIN {X 0,Y 258.898,Z 693.357,A -85,B 0,C 180,E1 12276.186,E2 12276.186} C_VEL
LIN {X 0,Y 262.043,Z 680.108,A -85,B 0,C 180,E1 12274.326,E2 12274.326} C_VEL
LIN {X 0,Y 264.995,Z 665.102,A -85,B 0,C 180,E1 12272.717,E2 12272.717} C_VEL
LIN {X 0,Y 267.294,Z 649.691,A -85,B 0,C 180,E1 12271.505,E2 12271.505} C_VEL
LIN {X 0,Y 268.986,Z 632.949,A -85,B 0,C 180,E1 12270.61,E2 12270.61} C_VEL
LIN {X 0,Y 270.617,Z 602.218,A -85,B 0,C 180,E1 12269.708,E2 12269.708} C_VEL
LIN {X 0,Y 275.313,Z 510.209,A -85,B 0,C 180,E1 12267.248,E2 12267.248} C_VEL
LIN {X 0,Y 273.512,Z 485.979,A -85,B 0,C 180,E1 12265.942,E2 12265.942} C_VEL
LIN {X 0,Y 280.045,Z 440.73,A -85,B 0,C 180,E1 12260.809,E2 12260.809} C_VEL
LIN {X 0,Y 286.282,Z 399.532,A -85,B 0,C 180,E1 12256.177,E2 12256.177} C_VEL
LIN {X 0,Y 287.247,Z 393.097,A -85,B 0,C 180,E1 12255.444,E2 12255.444} C_VEL
LIN {X 0,Y 283.992,Z 380.77,A -85,B 0,C 180,E1 12252.609,E2 12252.609} C_VEL
LIN {X 0,Y 280.11,Z 369.196,A -85,B 0,C 180,E1 12249.451,E2 12249.451} C_VEL
LIN {X 0,Y 275.927,Z 358.91,A -85,B 0,C 180,E1 12246.033,E2 12246.033} C_VEL
LIN {X 0,Y 272.236,Z 350.875,A -85,B 0,C 180,E1 12242.737,E2 12242.737} C_VEL
LIN {X 0,Y 269.55,Z 345.877,A -85,B 0,C 180,E1 12240.213,E2 12240.213} C_VEL
LIN {X 0,Y 267.534,Z 341.803,A -85,B 0,C 180,E1 12237.859,E2 12237.859} C_VEL
LIN {X 0,Y 265.369,Z 337.748,A -85,B 0,C 180,E1 12235.029,E2 12235.029} C_VEL
LIN {X 0,Y 264.4,Z 336.5,A -85,B 0,C 180,E1 12233.705,E2 12233.705} C_VEL
LIN {X 0,Y 262.185,Z 331.841,A -85,B 0,C 180,E1 12228.563,E2 12228.563} C_VEL
LIN {X 0,Y 261.185,Z 330.989,A -85,B 0,C 180,E1 12222.627,E2 12222.627} C_VEL
LIN {X 0,Y 262.323,Z 331.785,A -85,B 0,C 180,E1 12217.832,E2 12217.832} C_VEL
LIN {X 0,Y 262.258,Z 336.015,A -85,B 0,C 180,E1 12215.662,E2 12215.662} C_VEL
LIN {X 0,Y 262.325,Z 340.027,A -85,B 0,C 180,E1 12214.004,E2 12214.004} C_VEL
LIN {X 0,Y 262.766,Z 341.877,A -85,B 0,C 180,E1 12213.412,E2 12213.412} C_VEL
LIN {X 0,Y 275.605,Z 362.845,A -85,B 0,C 180,E1 12209.446,E2 12209.446} C_VEL
LIN {X 0,Y 288.747,Z 385.611,A -85,B 0,C 180,E1 12205.818,E2 12205.818} C_VEL
LIN {X 0,Y 298.163,Z 403.236,A -85,B 0,C 180,E1 12203.406,E2 12203.406} C_VEL
LIN {X 0,Y 281.724,Z 575.658,A -85,B 0,C 180,E1 12197.735,E2 12197.735} C_VEL
LIN {X 0,Y 278.71,Z 597.541,A -85,B 0,C 180,E1 12196.661,E2 12196.661} C_VEL
LIN {X 0,Y 275.124,Z 618.407,A -85,B 0,C 180,E1 12195.271,E2 12195.271} C_VEL
LIN {X 0,Y 270.941,Z 639.009,A -85,B 0,C 180,E1 12193.487,E2 12193.487} C_VEL
LIN {X 0,Y 266.524,Z 658.262,A -85,B 0,C 180,E1 12191.385,E2 12191.385} C_VEL
LIN {X 0,Y 261.89,Z 676.708,A -85,B 0,C 180,E1 12188.888,E2 12188.888} C_VEL
LIN {X 0,Y 257.448,Z 693.416,A -85,B 0,C 180,E1 12186.118,E2 12186.118} C_VEL
LIN {X 0,Y 253.07,Z 709.33,A -85,B 0,C 180,E1 12182.902,E2 12182.902} C_VEL
LIN {X 0,Y 249.3,Z 723.174,A -85,B 0,C 180,E1 12179.506,E2 12179.506} C_VEL
LIN {X 0,Y 246.038,Z 735.711,A -85,B 0,C 180,E1 12175.771,E2 12175.771} C_VEL
LIN {X 0,Y 243.824,Z 745.568,A -85,B 0,C 180,E1 12172.415,E2 12172.415} C_VEL
LIN {X 0,Y 242.235,Z 754.919,A -85,B 0,C 180,E1 12169.028,E2 12169.028} C_VEL
LIN {X 0,Y 241.07,Z 762.731,A -85,B 0,C 180,E1 12165.391,E2 12165.391} C_VEL
LIN {X 0,Y 240.415,Z 768.58,A -85,B 0,C 180,E1 12161.756,E2 12161.756} C_VEL
LIN {X 0,Y 240.179,Z 772.874,A -85,B 0,C 180,E1 12157.893,E2 12157.893} C_VEL
LIN {X 0,Y 240.196,Z 775.247,A -85,B 0,C 180,E1 12154.294,E2 12154.294} C_VEL
LIN {X 0,Y 240.275,Z 776.015,A -85,B 0,C 180,E1 12150.713,E2 12150.713} C_VEL
LIN {X 0,Y 240.208,Z 775.827,A -85,B 0,C 180,E1 12146.896,E2 12146.896} C_VEL
LIN {X 0,Y 240.081,Z 775.292,A -85,B 0,C 180,E1 12142.82,E2 12142.82} C_VEL
LIN {X 0,Y 240.332,Z 773.094,A -85,B 0,C 180,E1 12138.235,E2 12138.235} C_VEL
LIN {X 0,Y 241.568,Z 768.888,A -85,B 0,C 180,E1 12133.156,E2 12133.156} C_VEL
LIN {X 0,Y 244.168,Z 762.817,A -85,B 0,C 180,E1 12128.119,E2 12128.119} C_VEL
LIN {X 0,Y 248.363,Z 754.893,A -85,B 0,C 180,E1 12123.197,E2 12123.197} C_VEL
LIN {X 0,Y 254.275,Z 745.109,A -85,B 0,C 180,E1 12118.465,E2 12118.465} C_VEL
LIN {X 0,Y 262.379,Z 732.889,A -85,B 0,C 180,E1 12113.793,E2 12113.793} C_VEL
LIN {X 0,Y 272.493,Z 718.725,A -85,B 0,C 180,E1 12109.496,E2 12109.496} C_VEL
LIN {X 0,Y 285.244,Z 702.064,A -85,B 0,C 180,E1 12105.486,E2 12105.486} C_VEL
LIN {X 0,Y 298.345,Z 686.007,A -85,B 0,C 180,E1 12102.418,E2 12102.418} C_VEL
LIN {X 0,Y 285.435,Z 700.019,A -85,B 0,C 180,E1 12099.347,E2 12099.347} C_VEL
LIN {X 0,Y 273.446,Z 713.571,A -85,B 0,C 180,E1 12095.547,E2 12095.547} C_VEL
LIN {X 0,Y 263.45,Z 725.221,A -85,B 0,C 180,E1 12091.328,E2 12091.328} C_VEL
LIN {X 0,Y 255.57,Z 734.646,A -85,B 0,C 180,E1 12086.871,E2 12086.871} C_VEL
LIN {X 0,Y 249.47,Z 742.124,A -85,B 0,C 180,E1 12082.131,E2 12082.131} C_VEL
LIN {X 0,Y 245.302,Z 747.328,A -85,B 0,C 180,E1 12077.48,E2 12077.48} C_VEL
LIN {X 0,Y 242.619,Z 750.632,A -85,B 0,C 180,E1 12072.857,E2 12072.857} C_VEL
LIN {X 0,Y 241.057,Z 752.219,A -85,B 0,C 180,E1 12068.106,E2 12068.106} C_VEL
LIN {X 0,Y 240.395,Z 752.015,A -85,B 0,C 180,E1 12063.576,E2 12063.576} C_VEL
LIN {X 0,Y 240.2,Z 750.233,A -85,B 0,C 180,E1 12059.284,E2 12059.284} C_VEL
LIN {X 0,Y 240.21,Z 747.067,A -85,B 0,C 180,E1 12055.224,E2 12055.224} C_VEL
LIN {X 0,Y 240.52,Z 742.34,A -85,B 0,C 180,E1 12051.151,E2 12051.151} C_VEL
LIN {X 0,Y 241.371,Z 735.455,A -85,B 0,C 180,E1 12046.83,E2 12046.83} C_VEL
LIN {X 0,Y 242.857,Z 727.042,A -85,B 0,C 180,E1 12042.756,E2 12042.756} C_VEL
LIN {X 0,Y 244.974,Z 717.208,A -85,B 0,C 180,E1 12038.95,E2 12038.95} C_VEL
LIN {X 0,Y 247.871,Z 705.176,A -85,B 0,C 180,E1 12035.18,E2 12035.18} C_VEL
LIN {X 0,Y 251.297,Z 691.714,A -85,B 0,C 180,E1 12031.739,E2 12031.739} C_VEL
LIN {X 0,Y 255.157,Z 676.643,A -85,B 0,C 180,E1 12028.588,E2 12028.588} C_VEL
LIN {X 0,Y 259.477,Z 659.25,A -85,B 0,C 180,E1 12025.63,E2 12025.63} C_VEL
LIN {X 0,Y 263.643,Z 641.466,A -85,B 0,C 180,E1 12023.186,E2 12023.186} C_VEL
LIN {X 0,Y 267.756,Z 622.179,A -85,B 0,C 180,E1 12021.055,E2 12021.055} C_VEL
